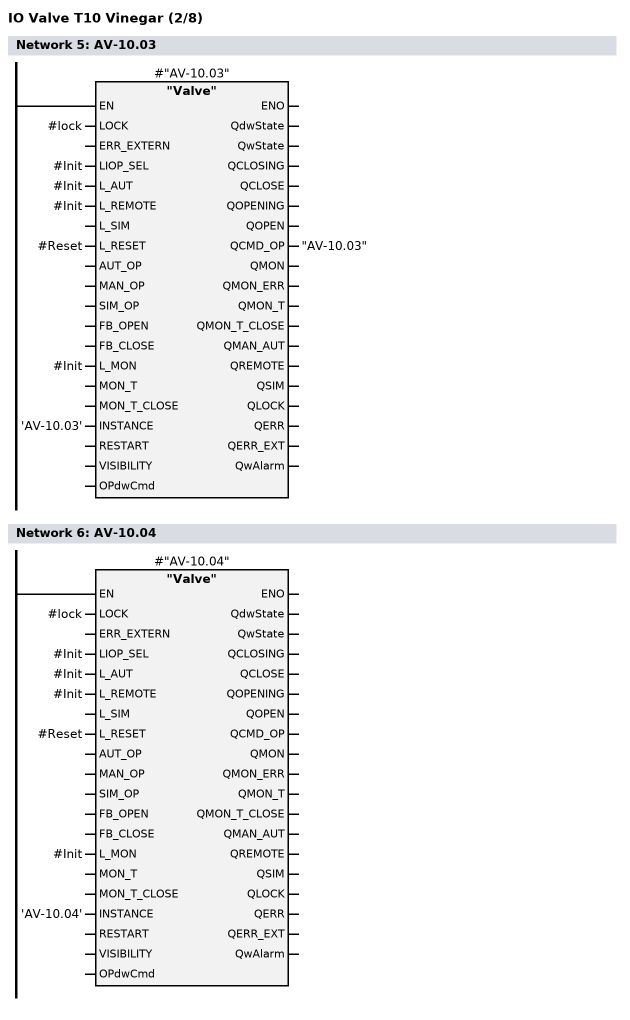
   RUNG wire#powerrail
      #"AV-10.03"(LOCK := #lock, ERR_EXTERN :=, LIOP_SEL := #Init, L_AUT := #Init, L_REMOTE := #Init, L_SIM :=, L_RESET := #Reset, AUT_OP :=, MAN_OP :=, SIM_OP :=, FB_OPEN :=, FB_CLOSE :=, L_MON := #Init, MON_T :=, MON_T_CLOSE :=, INSTANCE := 'AV-10.03', RESTART :=, VISIBILITY :=, OPdwCmd :=, QdwState =>, QwState =>, QCLOSING =>, QCLOSE =>, QOPENING =>, QOPEN =>, QCMD_OP => "AV-10.03", QMON =>, QMON_ERR =>, QMON_T =>, QMON_T_CLOSE =>, QMAN_AUT =>, QREMOTE =>, QSIM =>, QLOCK =>, QERR =>, QERR_EXT =>, QwAlarm =>)
   END_RUNG
   // the same network as SCL:
   #"AV-10.03"(LOCK := #lock,   // "Valve"
               LIOP_SEL := #Init,
               L_AUT := #Init,
               L_REMOTE := #Init,
               L_RESET := #Reset,
               L_MON := #Init,
               INSTANCE := 'AV-10.03',
               QCMD_OP => "AV-10.03");
END_REGION

REGION Network 6: AV-10.04
   RUNG wire#powerrail
      #"AV-10.04"(LOCK := #lock, ERR_EXTERN :=, LIOP_SEL := #Init, L_AUT := #Init, L_REMOTE := #Init, L_SIM :=, L_RESET := #Reset, AUT_OP :=, MAN_OP :=, SIM_OP :=, FB_OPEN :=, FB_CLOSE :=, L_MON := #Init, MON_T :=, MON_T_CLOSE :=, INSTANCE := 'AV-10.04', RESTART :=, VISIBILITY :=, OPdwCmd :=, QdwState =>, QwState =>, QCLOSING =>, QCLOSE =>, QOPENING =>, QOPEN =>, QCMD_OP =>, QMON =>, QMON_ERR =>, QMON_T =>, QMON_T_CLOSE =>, QMAN_AUT =>, QREMOTE =>, QSIM =>, QLOCK =>, QERR =>, QERR_EXT =>, QwAlarm =>)
   END_RUNG
   // the same network as SCL:
   #"AV-10.04"(LOCK := #lock,   // "Valve"
               LIOP_SEL := #Init,
               L_AUT := #Init,
               L_REMOTE := #Init,
               L_RESET := #Reset,
               L_MON := #Init,
               INSTANCE := 'AV-10.04');
END_REGION

REGION Network 7: AV-10.05
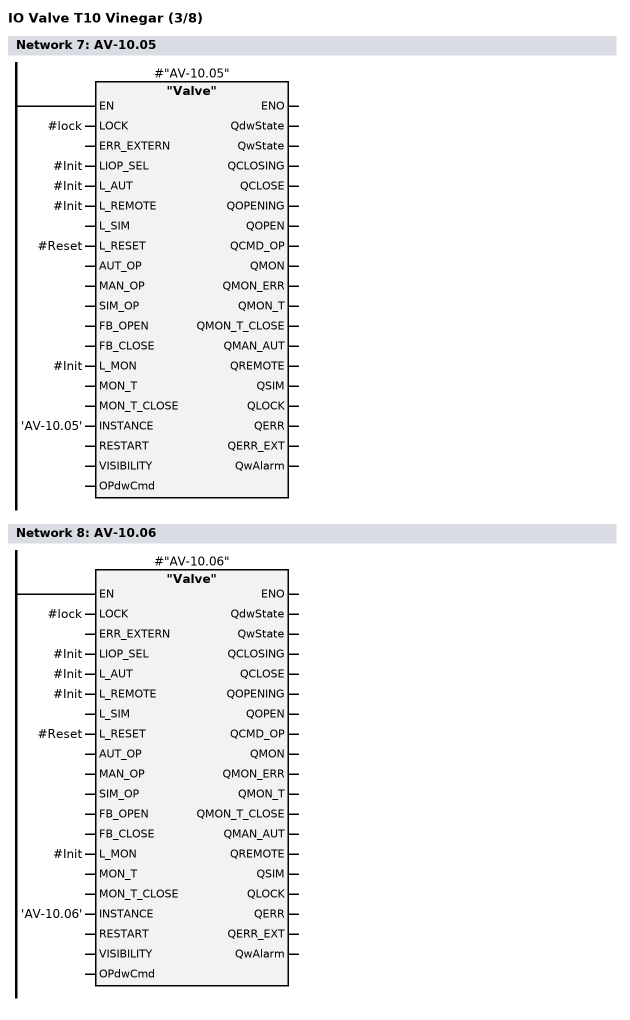
   RUNG wire#powerrail
      #"AV-10.05"(LOCK := #lock, ERR_EXTERN :=, LIOP_SEL := #Init, L_AUT := #Init, L_REMOTE := #Init, L_SIM :=, L_RESET := #Reset, AUT_OP :=, MAN_OP :=, SIM_OP :=, FB_OPEN :=, FB_CLOSE :=, L_MON := #Init, MON_T :=, MON_T_CLOSE :=, INSTANCE := 'AV-10.05', RESTART :=, VISIBILITY :=, OPdwCmd :=, QdwState =>, QwState =>, QCLOSING =>, QCLOSE =>, QOPENING =>, QOPEN =>, QCMD_OP =>, QMON =>, QMON_ERR =>, QMON_T =>, QMON_T_CLOSE =>, QMAN_AUT =>, QREMOTE =>, QSIM =>, QLOCK =>, QERR =>, QERR_EXT =>, QwAlarm =>)
   END_RUNG
   // the same network as SCL:
   #"AV-10.05"(LOCK := #lock,   // "Valve"
               LIOP_SEL := #Init,
               L_AUT := #Init,
               L_REMOTE := #Init,
               L_RESET := #Reset,
               L_MON := #Init,
               INSTANCE := 'AV-10.05');
END_REGION

REGION Network 8: AV-10.06
   RUNG wire#powerrail
      #"AV-10.06"(LOCK := #lock, ERR_EXTERN :=, LIOP_SEL := #Init, L_AUT := #Init, L_REMOTE := #Init, L_SIM :=, L_RESET := #Reset, AUT_OP :=, MAN_OP :=, SIM_OP :=, FB_OPEN :=, FB_CLOSE :=, L_MON := #Init, MON_T :=, MON_T_CLOSE :=, INSTANCE := 'AV-10.06', RESTART :=, VISIBILITY :=, OPdwCmd :=, QdwState =>, QwState =>, QCLOSING =>, QCLOSE =>, QOPENING =>, QOPEN =>, QCMD_OP =>, QMON =>, QMON_ERR =>, QMON_T =>, QMON_T_CLOSE =>, QMAN_AUT =>, QREMOTE =>, QSIM =>, QLOCK =>, QERR =>, QERR_EXT =>, QwAlarm =>)
   END_RUNG
   // the same network as SCL:
   #"AV-10.06"(LOCK := #lock,   // "Valve"
               LIOP_SEL := #Init,
               L_AUT := #Init,
               L_REMOTE := #Init,
               L_RESET := #Reset,
               L_MON := #Init,
               INSTANCE := 'AV-10.06');
END_REGION

REGION Network 9: AV-10.07
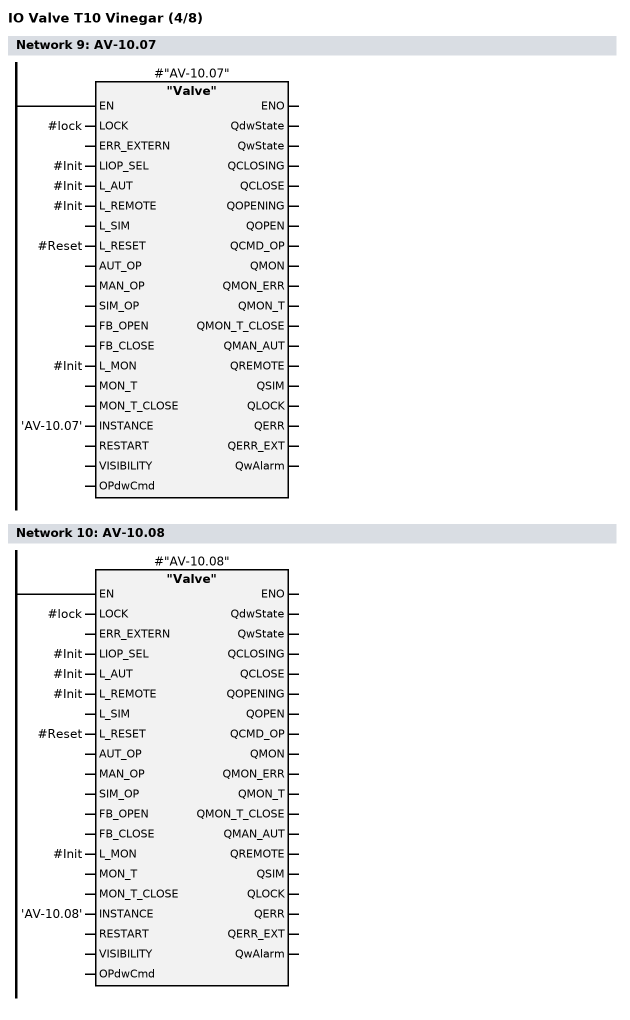
   RUNG wire#powerrail
      #"AV-10.07"(LOCK := #lock, ERR_EXTERN :=, LIOP_SEL := #Init, L_AUT := #Init, L_REMOTE := #Init, L_SIM :=, L_RESET := #Reset, AUT_OP :=, MAN_OP :=, SIM_OP :=, FB_OPEN :=, FB_CLOSE :=, L_MON := #Init, MON_T :=, MON_T_CLOSE :=, INSTANCE := 'AV-10.07', RESTART :=, VISIBILITY :=, OPdwCmd :=, QdwState =>, QwState =>, QCLOSING =>, QCLOSE =>, QOPENING =>, QOPEN =>, QCMD_OP =>, QMON =>, QMON_ERR =>, QMON_T =>, QMON_T_CLOSE =>, QMAN_AUT =>, QREMOTE =>, QSIM =>, QLOCK =>, QERR =>, QERR_EXT =>, QwAlarm =>)
   END_RUNG
   // the same network as SCL:
   #"AV-10.07"(LOCK := #lock,   // "Valve"
               LIOP_SEL := #Init,
               L_AUT := #Init,
               L_REMOTE := #Init,
               L_RESET := #Reset,
               L_MON := #Init,
               INSTANCE := 'AV-10.07');
END_REGION

REGION Network 10: AV-10.08
   RUNG wire#powerrail
      #"AV-10.08"(LOCK := #lock, ERR_EXTERN :=, LIOP_SEL := #Init, L_AUT := #Init, L_REMOTE := #Init, L_SIM :=, L_RESET := #Reset, AUT_OP :=, MAN_OP :=, SIM_OP :=, FB_OPEN :=, FB_CLOSE :=, L_MON := #Init, MON_T :=, MON_T_CLOSE :=, INSTANCE := 'AV-10.08', RESTART :=, VISIBILITY :=, OPdwCmd :=, QdwState =>, QwState =>, QCLOSING =>, QCLOSE =>, QOPENING =>, QOPEN =>, QCMD_OP =>, QMON =>, QMON_ERR =>, QMON_T =>, QMON_T_CLOSE =>, QMAN_AUT =>, QREMOTE =>, QSIM =>, QLOCK =>, QERR =>, QERR_EXT =>, QwAlarm =>)
   END_RUNG
   // the same network as SCL:
   #"AV-10.08"(LOCK := #lock,   // "Valve"
               LIOP_SEL := #Init,
               L_AUT := #Init,
               L_REMOTE := #Init,
               L_RESET := #Reset,
               L_MON := #Init,
               INSTANCE := 'AV-10.08');
END_REGION

REGION Network 11: AV-10.09
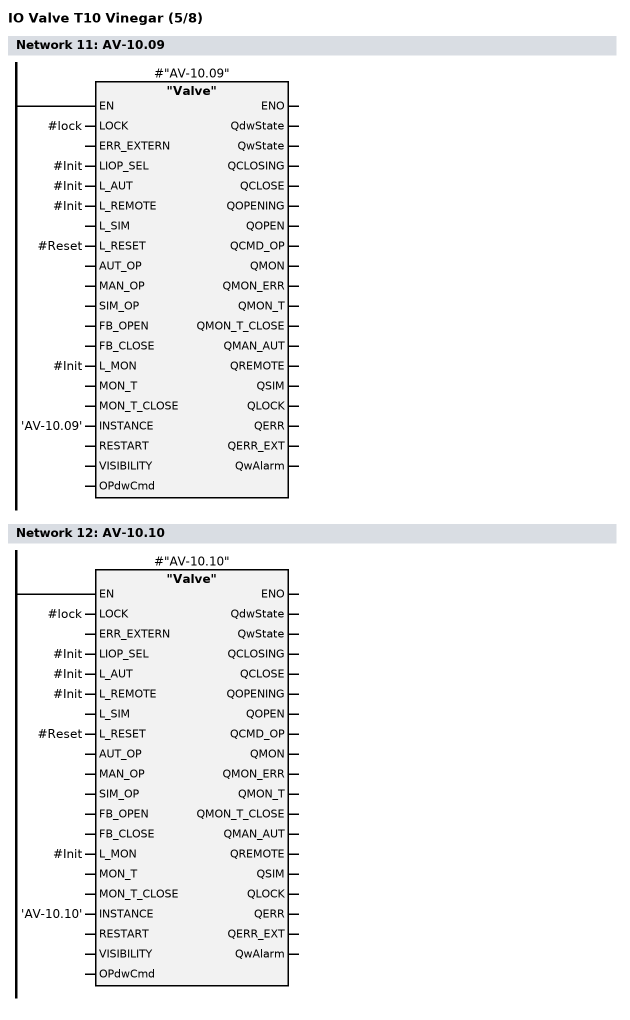
   RUNG wire#powerrail
      #"AV-10.09"(LOCK := #lock, ERR_EXTERN :=, LIOP_SEL := #Init, L_AUT := #Init, L_REMOTE := #Init, L_SIM :=, L_RESET := #Reset, AUT_OP :=, MAN_OP :=, SIM_OP :=, FB_OPEN :=, FB_CLOSE :=, L_MON := #Init, MON_T :=, MON_T_CLOSE :=, INSTANCE := 'AV-10.09', RESTART :=, VISIBILITY :=, OPdwCmd :=, QdwState =>, QwState =>, QCLOSING =>, QCLOSE =>, QOPENING =>, QOPEN =>, QCMD_OP =>, QMON =>, QMON_ERR =>, QMON_T =>, QMON_T_CLOSE =>, QMAN_AUT =>, QREMOTE =>, QSIM =>, QLOCK =>, QERR =>, QERR_EXT =>, QwAlarm =>)
   END_RUNG
   // the same network as SCL:
   #"AV-10.09"(LOCK := #lock,   // "Valve"
               LIOP_SEL := #Init,
               L_AUT := #Init,
               L_REMOTE := #Init,
               L_RESET := #Reset,
               L_MON := #Init,
               INSTANCE := 'AV-10.09');
END_REGION

REGION Network 12: AV-10.10
   RUNG wire#powerrail
      #"AV-10.10"(LOCK := #lock, ERR_EXTERN :=, LIOP_SEL := #Init, L_AUT := #Init, L_REMOTE := #Init, L_SIM :=, L_RESET := #Reset, AUT_OP :=, MAN_OP :=, SIM_OP :=, FB_OPEN :=, FB_CLOSE :=, L_MON := #Init, MON_T :=, MON_T_CLOSE :=, INSTANCE := 'AV-10.10', RESTART :=, VISIBILITY :=, OPdwCmd :=, QdwState =>, QwState =>, QCLOSING =>, QCLOSE =>, QOPENING =>, QOPEN =>, QCMD_OP =>, QMON =>, QMON_ERR =>, QMON_T =>, QMON_T_CLOSE =>, QMAN_AUT =>, QREMOTE =>, QSIM =>, QLOCK =>, QERR =>, QERR_EXT =>, QwAlarm =>)
   END_RUNG
   // the same network as SCL:
   #"AV-10.10"(LOCK := #lock,   // "Valve"
               LIOP_SEL := #Init,
               L_AUT := #Init,
               L_REMOTE := #Init,
               L_RESET := #Reset,
               L_MON := #Init,
               INSTANCE := 'AV-10.10');
END_REGION

REGION Network 13: AV-10.11
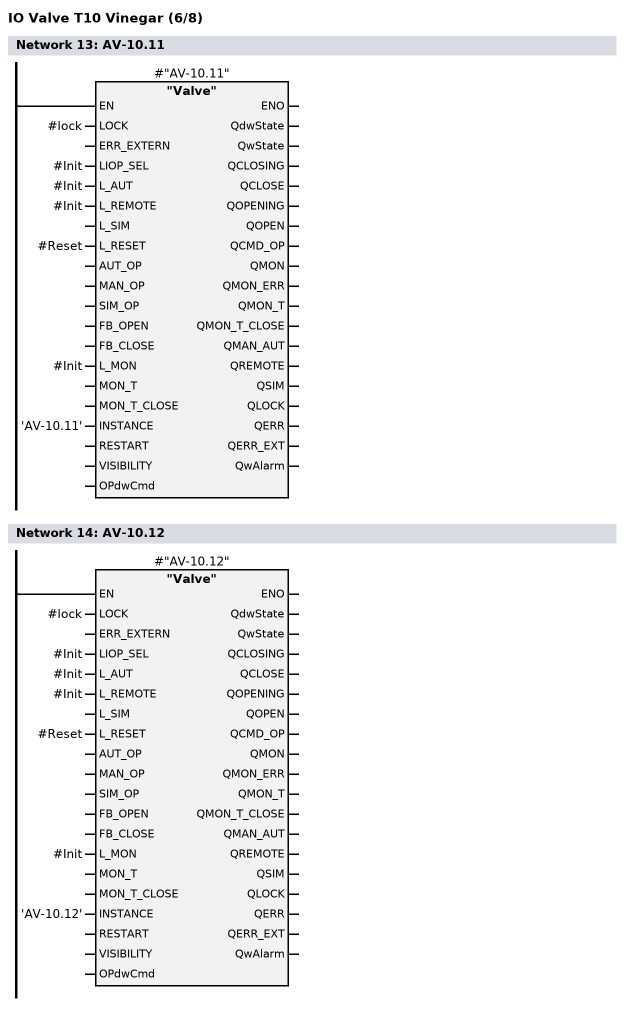
   RUNG wire#powerrail
      #"AV-10.11"(LOCK := #lock, ERR_EXTERN :=, LIOP_SEL := #Init, L_AUT := #Init, L_REMOTE := #Init, L_SIM :=, L_RESET := #Reset, AUT_OP :=, MAN_OP :=, SIM_OP :=, FB_OPEN :=, FB_CLOSE :=, L_MON := #Init, MON_T :=, MON_T_CLOSE :=, INSTANCE := 'AV-10.11', RESTART :=, VISIBILITY :=, OPdwCmd :=, QdwState =>, QwState =>, QCLOSING =>, QCLOSE =>, QOPENING =>, QOPEN =>, QCMD_OP =>, QMON =>, QMON_ERR =>, QMON_T =>, QMON_T_CLOSE =>, QMAN_AUT =>, QREMOTE =>, QSIM =>, QLOCK =>, QERR =>, QERR_EXT =>, QwAlarm =>)
   END_RUNG
   // the same network as SCL:
   #"AV-10.11"(LOCK := #lock,   // "Valve"
               LIOP_SEL := #Init,
               L_AUT := #Init,
               L_REMOTE := #Init,
               L_RESET := #Reset,
               L_MON := #Init,
               INSTANCE := 'AV-10.11');
END_REGION

REGION Network 14: AV-10.12
   RUNG wire#powerrail
      #"AV-10.12"(LOCK := #lock, ERR_EXTERN :=, LIOP_SEL := #Init, L_AUT := #Init, L_REMOTE := #Init, L_SIM :=, L_RESET := #Reset, AUT_OP :=, MAN_OP :=, SIM_OP :=, FB_OPEN :=, FB_CLOSE :=, L_MON := #Init, MON_T :=, MON_T_CLOSE :=, INSTANCE := 'AV-10.12', RESTART :=, VISIBILITY :=, OPdwCmd :=, QdwState =>, QwState =>, QCLOSING =>, QCLOSE =>, QOPENING =>, QOPEN =>, QCMD_OP =>, QMON =>, QMON_ERR =>, QMON_T =>, QMON_T_CLOSE =>, QMAN_AUT =>, QREMOTE =>, QSIM =>, QLOCK =>, QERR =>, QERR_EXT =>, QwAlarm =>)
   END_RUNG
   // the same network as SCL:
   #"AV-10.12"(LOCK := #lock,   // "Valve"
               LIOP_SEL := #Init,
               L_AUT := #Init,
               L_REMOTE := #Init,
               L_RESET := #Reset,
               L_MON := #Init,
               INSTANCE := 'AV-10.12');
END_REGION

REGION Network 15: AV-10.13
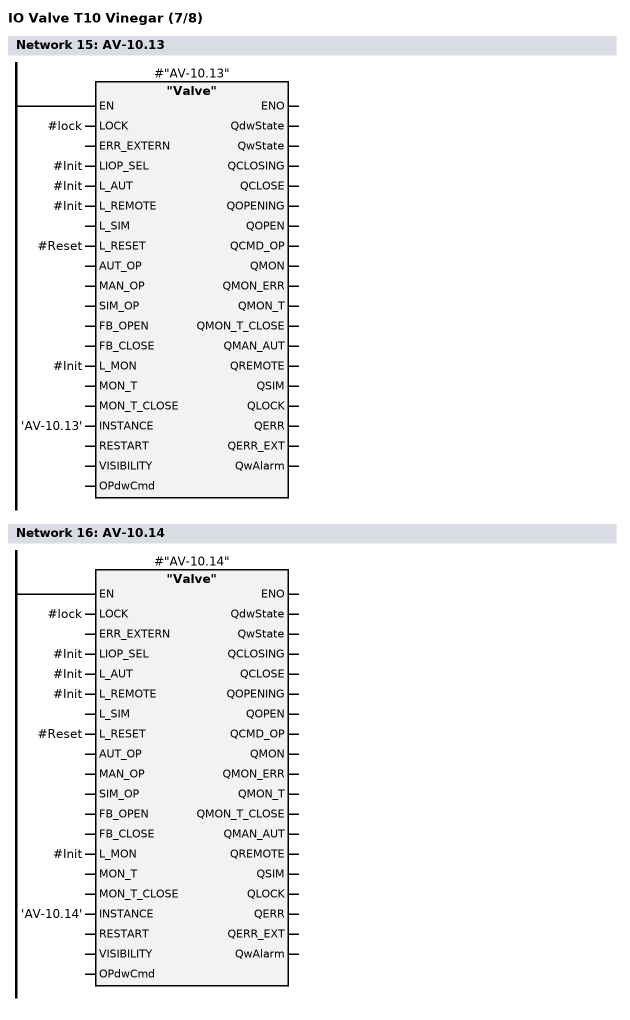
   RUNG wire#powerrail
      #"AV-10.13"(LOCK := #lock, ERR_EXTERN :=, LIOP_SEL := #Init, L_AUT := #Init, L_REMOTE := #Init, L_SIM :=, L_RESET := #Reset, AUT_OP :=, MAN_OP :=, SIM_OP :=, FB_OPEN :=, FB_CLOSE :=, L_MON := #Init, MON_T :=, MON_T_CLOSE :=, INSTANCE := 'AV-10.13', RESTART :=, VISIBILITY :=, OPdwCmd :=, QdwState =>, QwState =>, QCLOSING =>, QCLOSE =>, QOPENING =>, QOPEN =>, QCMD_OP =>, QMON =>, QMON_ERR =>, QMON_T =>, QMON_T_CLOSE =>, QMAN_AUT =>, QREMOTE =>, QSIM =>, QLOCK =>, QERR =>, QERR_EXT =>, QwAlarm =>)
   END_RUNG
   // the same network as SCL:
   #"AV-10.13"(LOCK := #lock,   // "Valve"
               LIOP_SEL := #Init,
               L_AUT := #Init,
               L_REMOTE := #Init,
               L_RESET := #Reset,
               L_MON := #Init,
               INSTANCE := 'AV-10.13');
END_REGION

REGION Network 16: AV-10.14
   RUNG wire#powerrail
      #"AV-10.14"(LOCK := #lock, ERR_EXTERN :=, LIOP_SEL := #Init, L_AUT := #Init, L_REMOTE := #Init, L_SIM :=, L_RESET := #Reset, AUT_OP :=, MAN_OP :=, SIM_OP :=, FB_OPEN :=, FB_CLOSE :=, L_MON := #Init, MON_T :=, MON_T_CLOSE :=, INSTANCE := 'AV-10.14', RESTART :=, VISIBILITY :=, OPdwCmd :=, QdwState =>, QwState =>, QCLOSING =>, QCLOSE =>, QOPENING =>, QOPEN =>, QCMD_OP =>, QMON =>, QMON_ERR =>, QMON_T =>, QMON_T_CLOSE =>, QMAN_AUT =>, QREMOTE =>, QSIM =>, QLOCK =>, QERR =>, QERR_EXT =>, QwAlarm =>)
   END_RUNG
   // the same network as SCL:
   #"AV-10.14"(LOCK := #lock,   // "Valve"
               LIOP_SEL := #Init,
               L_AUT := #Init,
               L_REMOTE := #Init,
               L_RESET := #Reset,
               L_MON := #Init,
               INSTANCE := 'AV-10.14');
END_REGION

REGION Network 17: P-10.02
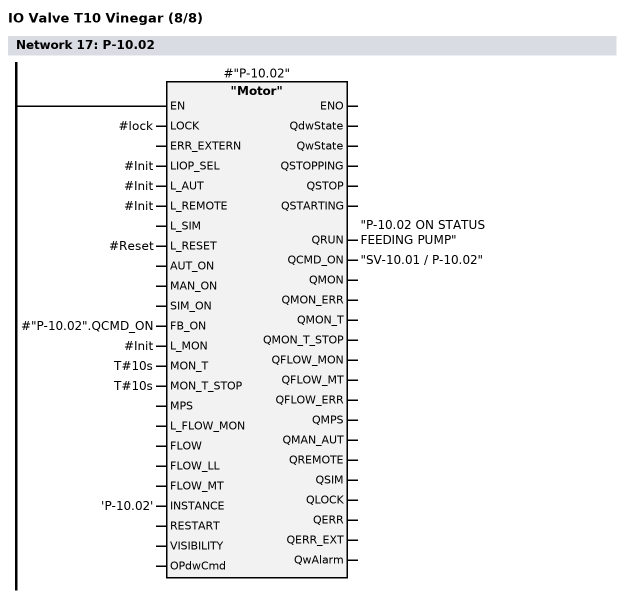
   RUNG wire#powerrail
      #"P-10.02"(LOCK := #lock, ERR_EXTERN :=, LIOP_SEL := #Init, L_AUT := #Init, L_REMOTE := #Init, L_SIM :=, L_RESET := #Reset, AUT_ON :=, MAN_ON :=, SIM_ON :=, FB_ON := #"P-10.02".QCMD_ON, L_MON := #Init, MON_T := T#10s, MON_T_STOP := T#10s, MPS :=, L_FLOW_MON :=, FLOW :=, FLOW_LL :=, FLOW_MT :=, INSTANCE := 'P-10.02', RESTART :=, VISIBILITY :=, OPdwCmd :=, QdwState =>, QwState =>, QSTOPPING =>, QSTOP =>, QSTARTING =>, QRUN => "P-10.02 ON STATUS FEEDING PUMP", QCMD_ON => "SV-10.01 / P-10.02", QMON =>, QMON_ERR =>, QMON_T =>, QMON_T_STOP =>, QFLOW_MON =>, QFLOW_MT =>, QFLOW_ERR =>, QMPS =>, QMAN_AUT =>, QREMOTE =>, QSIM =>, QLOCK =>, QERR =>, QERR_EXT =>, QwAlarm =>)
   END_RUNG
   // the same network as SCL:
   #"P-10.02"(LOCK := #lock,   // "Motor"
              LIOP_SEL := #Init,
              L_AUT := #Init,
              L_REMOTE := #Init,
              L_RESET := #Reset,
              FB_ON := #"P-10.02".QCMD_ON,
              L_MON := #Init,
              MON_T := T#10s,
              MON_T_STOP := T#10s,
              INSTANCE := 'P-10.02',
              QRUN => "P-10.02 ON STATUS FEEDING PUMP",
              QCMD_ON => "SV-10.01 / P-10.02");
END_REGION
END_FUNCTION_BLOCK

FUNCTION_BLOCK "IO Valve T51 HotWaterLine"   // FB311, LAD
{ S7_Optimized_Access := 'FALSE' }
VERSION : 0.1
// stored: AutoNumber false, IsIECCheckEnabled false, SetENOAutomatically false, UDAEnableTagReadback false
   VAR_INPUT
      lock : Bool;
      Init : Bool;
      testing : Bool;
      Reset : Bool;
   END_VAR
   VAR
      "AV-51.01" { S7_SetPoint := 'True'} : "Valve";
      "AV-51.02" { S7_SetPoint := 'True'} : "Valve";
      "AV-51.03" { S7_SetPoint := 'True'} : "Valve";
      "AV-51.04" { S7_SetPoint := 'True'} : "Valve";
      "AV-51.05" { S7_SetPoint := 'True'} : "Valve";
      "AV-51.06" { S7_SetPoint := 'True'} : "Valve";
      "AV-51.07" { S7_SetPoint := 'True'} : "Valve";
      "AV-51.08" { S7_SetPoint := 'True'} : "Valve";
      "AV-51.09" { S7_SetPoint := 'True'} : "Valve";
      "AV-51.10" { S7_SetPoint := 'True'} : "Valve";
      "AV-51.11" { S7_SetPoint := 'True'} : "Valve";
      "AV-51.12" { S7_SetPoint := 'True'} : "Valve";
      "AV-51.13" { S7_SetPoint := 'True'} : "Valve";
      "AV-51.14" { S7_SetPoint := 'True'} : "Valve";
      "AV-51.15" { S7_SetPoint := 'True'} : "Valve";
      "CV-51.11" { S7_SetPoint := 'True'} : "Valve";
   END_VAR
BEGIN

REGION Network 1 (SCL): FB OPEN and CLOSE
   IF #testing THEN
       // Statement section IF
       #"AV-51.01".FB_OPEN := #"AV-51.01".QCMD_OP;
       #"AV-51.01".FB_CLOSE := NOT #"AV-51.01".QCMD_OP;
       #"AV-51.02".FB_OPEN := #"AV-51.02".QCMD_OP;
       #"AV-51.02".FB_CLOSE := NOT #"AV-51.02".QCMD_OP;
       #"AV-51.03".FB_OPEN := #"AV-51.03".QCMD_OP;
       #"AV-51.03".FB_CLOSE := NOT #"AV-51.03".QCMD_OP;
       #"AV-51.04".FB_OPEN := #"AV-51.04".QCMD_OP;
       #"AV-51.04".FB_CLOSE := NOT #"AV-51.04".QCMD_OP;
       #"AV-51.05".FB_OPEN := #"AV-51.05".QCMD_OP;
       #"AV-51.05".FB_CLOSE := NOT #"AV-51.05".QCMD_OP;
       #"AV-51.06".FB_OPEN := #"AV-51.06".QCMD_OP;
       #"AV-51.06".FB_CLOSE := NOT #"AV-51.06".QCMD_OP;
       #"AV-51.07".FB_OPEN := #"AV-51.07".QCMD_OP;
       #"AV-51.07".FB_CLOSE := NOT #"AV-51.07".QCMD_OP;
       #"AV-51.08".FB_OPEN := #"AV-51.08".QCMD_OP;
       #"AV-51.08".FB_CLOSE := NOT #"AV-51.08".QCMD_OP;
       #"AV-51.09".FB_OPEN := #"AV-51.09".QCMD_OP;
       #"AV-51.09".FB_CLOSE := NOT #"AV-51.09".QCMD_OP;
       #"AV-51.10".FB_OPEN := #"AV-51.10".QCMD_OP;
       #"AV-51.10".FB_CLOSE := NOT #"AV-51.10".QCMD_OP;
       #"AV-51.11".FB_OPEN := #"AV-51.11".QCMD_OP;
       #"AV-51.11".FB_CLOSE := NOT #"AV-51.11".QCMD_OP;
       #"AV-51.12".FB_OPEN := #"AV-51.12".QCMD_OP;
       #"AV-51.12".FB_CLOSE := NOT #"AV-51.12".QCMD_OP;
       #"AV-51.13".FB_OPEN := #"AV-51.13".QCMD_OP;
       #"AV-51.13".FB_CLOSE := NOT #"AV-51.13".QCMD_OP;
       #"AV-51.14".FB_OPEN := #"AV-51.14".QCMD_OP;
       #"AV-51.14".FB_CLOSE := NOT #"AV-51.14".QCMD_OP;
       #"AV-51.15".FB_OPEN := #"AV-51.15".QCMD_OP;
       #"AV-51.15".FB_CLOSE := NOT #"AV-51.15".QCMD_OP;
   ELSE
       // Statement section ELSE
       #"AV-51.01".FB_OPEN := #"AV-51.01".QCMD_OP;
       #"AV-51.01".FB_CLOSE := NOT #"AV-51.01".QCMD_OP;
       #"AV-51.02".FB_OPEN := #"AV-51.02".QCMD_OP;
       #"AV-51.02".FB_CLOSE := NOT #"AV-51.02".QCMD_OP;
       #"AV-51.03".FB_OPEN := #"AV-51.03".QCMD_OP;
       #"AV-51.03".FB_CLOSE := NOT #"AV-51.03".QCMD_OP;
       #"AV-51.04".FB_OPEN := NOT "ZSC-51.04";
       #"AV-51.04".FB_CLOSE := "ZSC-51.04";
       #"AV-51.05".FB_OPEN := NOT "ZSC-51.05";
       #"AV-51.05".FB_CLOSE := "ZSC-51.05";
       #"AV-51.06".FB_OPEN := #"AV-51.06".QCMD_OP;
       #"AV-51.06".FB_CLOSE := NOT #"AV-51.06".QCMD_OP;
       #"AV-51.07".FB_OPEN := #"AV-51.07".QCMD_OP;
       #"AV-51.07".FB_CLOSE := NOT #"AV-51.07".QCMD_OP;
       #"AV-51.08".FB_OPEN := #"AV-51.08".QCMD_OP;
       #"AV-51.08".FB_CLOSE := NOT #"AV-51.08".QCMD_OP;
       #"AV-51.09".FB_OPEN := #"AV-51.09".QCMD_OP;
       #"AV-51.09".FB_CLOSE := NOT #"AV-51.09".QCMD_OP;
       #"AV-51.10".FB_OPEN := #"AV-51.10".QCMD_OP;
       #"AV-51.10".FB_CLOSE := NOT #"AV-51.10".QCMD_OP;
       #"AV-51.11".FB_OPEN := #"AV-51.11".QCMD_OP;
       #"AV-51.11".FB_CLOSE := NOT #"AV-51.11".QCMD_OP;
       #"AV-51.12".FB_OPEN := #"AV-51.12".QCMD_OP;
       #"AV-51.12".FB_CLOSE := NOT #"AV-51.12".QCMD_OP;
       #"AV-51.13".FB_OPEN := #"AV-51.13".QCMD_OP;
       #"AV-51.13".FB_CLOSE := NOT #"AV-51.13".QCMD_OP;
       #"AV-51.14".FB_OPEN := #"AV-51.14".QCMD_OP;
       #"AV-51.14".FB_CLOSE := NOT #"AV-51.14".QCMD_OP;
       #"AV-51.15".FB_OPEN := #"AV-51.15".QCMD_OP;
       #"AV-51.15".FB_CLOSE := NOT #"AV-51.15".QCMD_OP;
   END_IF;
END_REGION

NETWORK
TITLE = FB Monitoring Time
// FB OPEN Time
      L     t#20s;
      T     #"AV-51.01".MON_T;
      T     #"AV-51.02".MON_T;
      T     #"AV-51.03".MON_T;
      T     #"AV-51.04".MON_T;
      T     #"AV-51.05".MON_T;
      T     #"AV-51.06".MON_T;
      T     #"AV-51.07".MON_T;
      T     #"AV-51.08".MON_T;
      T     #"AV-51.09".MON_T;
      T     #"AV-51.10".MON_T;
      T     #"AV-51.11".MON_T;
      T     #"AV-51.12".MON_T;
      T     #"AV-51.13".MON_T;
      T     #"AV-51.14".MON_T;
      T     #"AV-51.15".MON_T;
// FB CLOSE Time
      L     t#20s;
      T     #"AV-51.01".MON_T_CLOSE;
      T     #"AV-51.02".MON_T_CLOSE;
      T     #"AV-51.03".MON_T_CLOSE;
      T     #"AV-51.04".MON_T_CLOSE;
      T     #"AV-51.05".MON_T_CLOSE;
      T     #"AV-51.06".MON_T_CLOSE;
      T     #"AV-51.07".MON_T_CLOSE;
      T     #"AV-51.08".MON_T_CLOSE;
      T     #"AV-51.09".MON_T_CLOSE;
      T     #"AV-51.10".MON_T_CLOSE;
      T     #"AV-51.11".MON_T_CLOSE;
      T     #"AV-51.12".MON_T_CLOSE;
      T     #"AV-51.13".MON_T_CLOSE;
      T     #"AV-51.14".MON_T_CLOSE;
      T     #"AV-51.15".MON_T_CLOSE;

REGION Network 3: AV-51.01
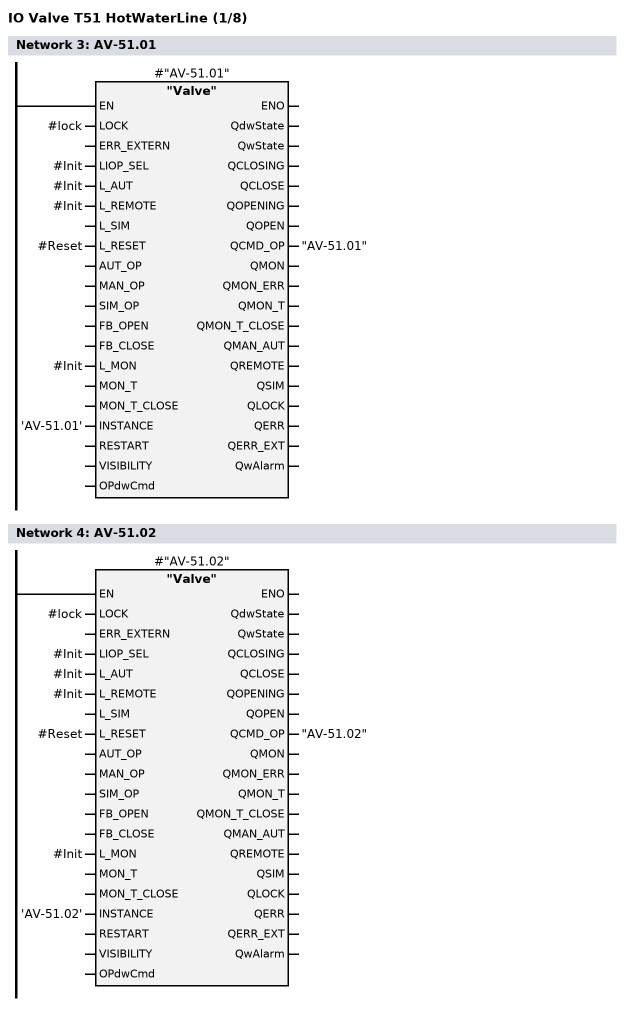
   RUNG wire#powerrail
      #"AV-51.01"(LOCK := #lock, ERR_EXTERN :=, LIOP_SEL := #Init, L_AUT := #Init, L_REMOTE := #Init, L_SIM :=, L_RESET := #Reset, AUT_OP :=, MAN_OP :=, SIM_OP :=, FB_OPEN :=, FB_CLOSE :=, L_MON := #Init, MON_T :=, MON_T_CLOSE :=, INSTANCE := 'AV-51.01', RESTART :=, VISIBILITY :=, OPdwCmd :=, QdwState =>, QwState =>, QCLOSING =>, QCLOSE =>, QOPENING =>, QOPEN =>, QCMD_OP => "AV-51.01", QMON =>, QMON_ERR =>, QMON_T =>, QMON_T_CLOSE =>, QMAN_AUT =>, QREMOTE =>, QSIM =>, QLOCK =>, QERR =>, QERR_EXT =>, QwAlarm =>)
   END_RUNG
   // the same network as SCL:
   #"AV-51.01"(LOCK := #lock,   // "Valve"
               LIOP_SEL := #Init,
               L_AUT := #Init,
               L_REMOTE := #Init,
               L_RESET := #Reset,
               L_MON := #Init,
               INSTANCE := 'AV-51.01',
               QCMD_OP => "AV-51.01");
END_REGION

REGION Network 4: AV-51.02
   RUNG wire#powerrail
      #"AV-51.02"(LOCK := #lock, ERR_EXTERN :=, LIOP_SEL := #Init, L_AUT := #Init, L_REMOTE := #Init, L_SIM :=, L_RESET := #Reset, AUT_OP :=, MAN_OP :=, SIM_OP :=, FB_OPEN :=, FB_CLOSE :=, L_MON := #Init, MON_T :=, MON_T_CLOSE :=, INSTANCE := 'AV-51.02', RESTART :=, VISIBILITY :=, OPdwCmd :=, QdwState =>, QwState =>, QCLOSING =>, QCLOSE =>, QOPENING =>, QOPEN =>, QCMD_OP => "AV-51.02", QMON =>, QMON_ERR =>, QMON_T =>, QMON_T_CLOSE =>, QMAN_AUT =>, QREMOTE =>, QSIM =>, QLOCK =>, QERR =>, QERR_EXT =>, QwAlarm =>)
   END_RUNG
   // the same network as SCL:
   #"AV-51.02"(LOCK := #lock,   // "Valve"
               LIOP_SEL := #Init,
               L_AUT := #Init,
               L_REMOTE := #Init,
               L_RESET := #Reset,
               L_MON := #Init,
               INSTANCE := 'AV-51.02',
               QCMD_OP => "AV-51.02");
END_REGION

REGION Network 5: AV-51.03
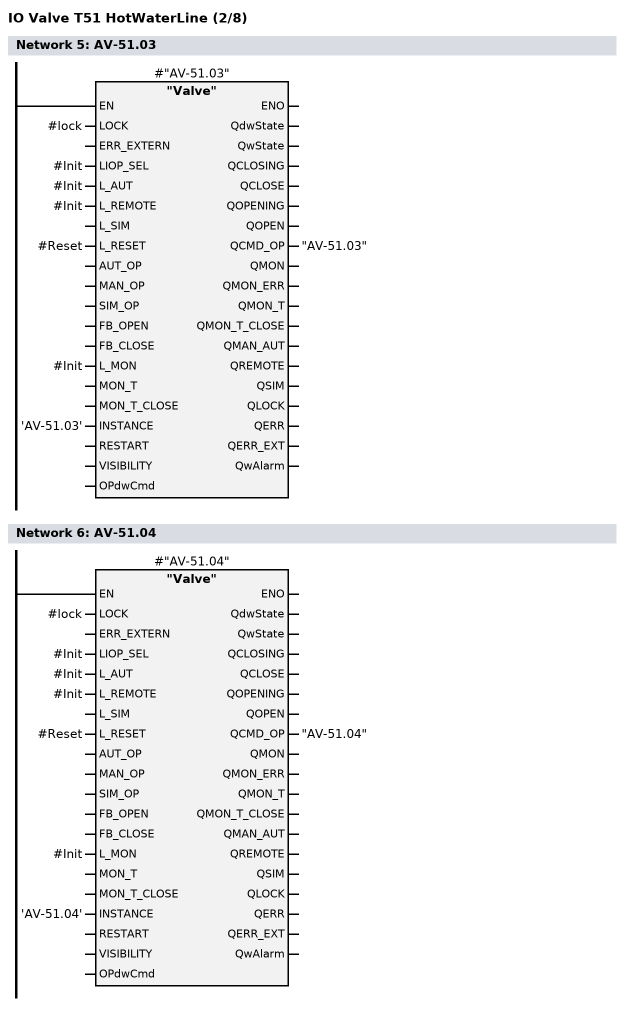
   RUNG wire#powerrail
      #"AV-51.03"(LOCK := #lock, ERR_EXTERN :=, LIOP_SEL := #Init, L_AUT := #Init, L_REMOTE := #Init, L_SIM :=, L_RESET := #Reset, AUT_OP :=, MAN_OP :=, SIM_OP :=, FB_OPEN :=, FB_CLOSE :=, L_MON := #Init, MON_T :=, MON_T_CLOSE :=, INSTANCE := 'AV-51.03', RESTART :=, VISIBILITY :=, OPdwCmd :=, QdwState =>, QwState =>, QCLOSING =>, QCLOSE =>, QOPENING =>, QOPEN =>, QCMD_OP => "AV-51.03", QMON =>, QMON_ERR =>, QMON_T =>, QMON_T_CLOSE =>, QMAN_AUT =>, QREMOTE =>, QSIM =>, QLOCK =>, QERR =>, QERR_EXT =>, QwAlarm =>)
   END_RUNG
   // the same network as SCL:
   #"AV-51.03"(LOCK := #lock,   // "Valve"
               LIOP_SEL := #Init,
               L_AUT := #Init,
               L_REMOTE := #Init,
               L_RESET := #Reset,
               L_MON := #Init,
               INSTANCE := 'AV-51.03',
               QCMD_OP => "AV-51.03");
END_REGION

REGION Network 6: AV-51.04
   RUNG wire#powerrail
      #"AV-51.04"(LOCK := #lock, ERR_EXTERN :=, LIOP_SEL := #Init, L_AUT := #Init, L_REMOTE := #Init, L_SIM :=, L_RESET := #Reset, AUT_OP :=, MAN_OP :=, SIM_OP :=, FB_OPEN :=, FB_CLOSE :=, L_MON := #Init, MON_T :=, MON_T_CLOSE :=, INSTANCE := 'AV-51.04', RESTART :=, VISIBILITY :=, OPdwCmd :=, QdwState =>, QwState =>, QCLOSING =>, QCLOSE =>, QOPENING =>, QOPEN =>, QCMD_OP => "AV-51.04", QMON =>, QMON_ERR =>, QMON_T =>, QMON_T_CLOSE =>, QMAN_AUT =>, QREMOTE =>, QSIM =>, QLOCK =>, QERR =>, QERR_EXT =>, QwAlarm =>)
   END_RUNG
   // the same network as SCL:
   #"AV-51.04"(LOCK := #lock,   // "Valve"
               LIOP_SEL := #Init,
               L_AUT := #Init,
               L_REMOTE := #Init,
               L_RESET := #Reset,
               L_MON := #Init,
               INSTANCE := 'AV-51.04',
               QCMD_OP => "AV-51.04");
END_REGION

REGION Network 7: AV-51.05
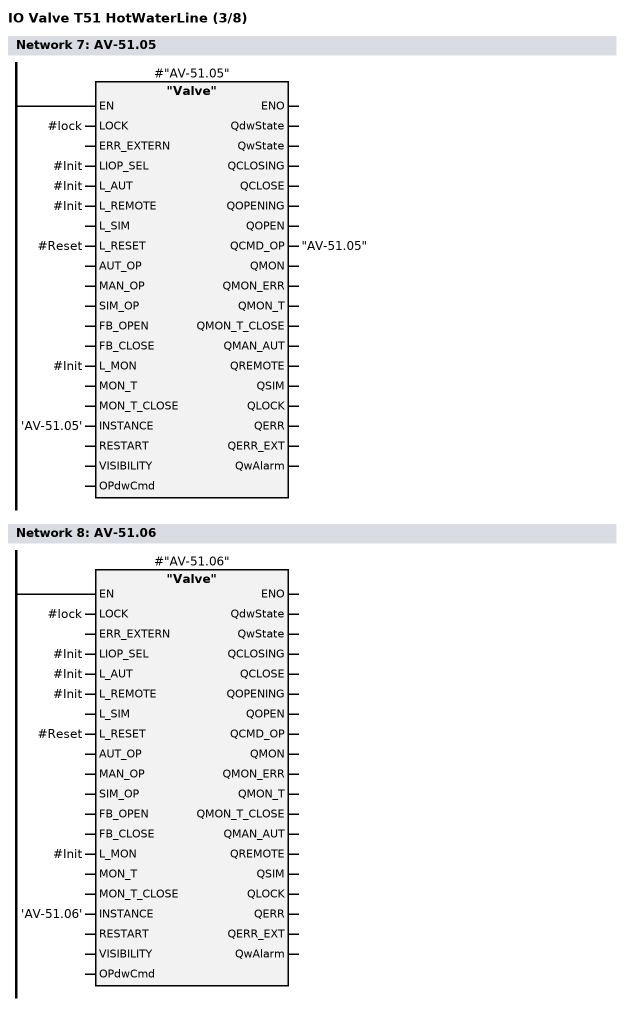
   RUNG wire#powerrail
      #"AV-51.05"(LOCK := #lock, ERR_EXTERN :=, LIOP_SEL := #Init, L_AUT := #Init, L_REMOTE := #Init, L_SIM :=, L_RESET := #Reset, AUT_OP :=, MAN_OP :=, SIM_OP :=, FB_OPEN :=, FB_CLOSE :=, L_MON := #Init, MON_T :=, MON_T_CLOSE :=, INSTANCE := 'AV-51.05', RESTART :=, VISIBILITY :=, OPdwCmd :=, QdwState =>, QwState =>, QCLOSING =>, QCLOSE =>, QOPENING =>, QOPEN =>, QCMD_OP => "AV-51.05", QMON =>, QMON_ERR =>, QMON_T =>, QMON_T_CLOSE =>, QMAN_AUT =>, QREMOTE =>, QSIM =>, QLOCK =>, QERR =>, QERR_EXT =>, QwAlarm =>)
   END_RUNG
   // the same network as SCL:
   #"AV-51.05"(LOCK := #lock,   // "Valve"
               LIOP_SEL := #Init,
               L_AUT := #Init,
               L_REMOTE := #Init,
               L_RESET := #Reset,
               L_MON := #Init,
               INSTANCE := 'AV-51.05',
               QCMD_OP => "AV-51.05");
END_REGION

REGION Network 8: AV-51.06
   RUNG wire#powerrail
      #"AV-51.06"(LOCK := #lock, ERR_EXTERN :=, LIOP_SEL := #Init, L_AUT := #Init, L_REMOTE := #Init, L_SIM :=, L_RESET := #Reset, AUT_OP :=, MAN_OP :=, SIM_OP :=, FB_OPEN :=, FB_CLOSE :=, L_MON := #Init, MON_T :=, MON_T_CLOSE :=, INSTANCE := 'AV-51.06', RESTART :=, VISIBILITY :=, OPdwCmd :=, QdwState =>, QwState =>, QCLOSING =>, QCLOSE =>, QOPENING =>, QOPEN =>, QCMD_OP =>, QMON =>, QMON_ERR =>, QMON_T =>, QMON_T_CLOSE =>, QMAN_AUT =>, QREMOTE =>, QSIM =>, QLOCK =>, QERR =>, QERR_EXT =>, QwAlarm =>)
   END_RUNG
   // the same network as SCL:
   #"AV-51.06"(LOCK := #lock,   // "Valve"
               LIOP_SEL := #Init,
               L_AUT := #Init,
               L_REMOTE := #Init,
               L_RESET := #Reset,
               L_MON := #Init,
               INSTANCE := 'AV-51.06');
END_REGION

REGION Network 9: AV-51.07
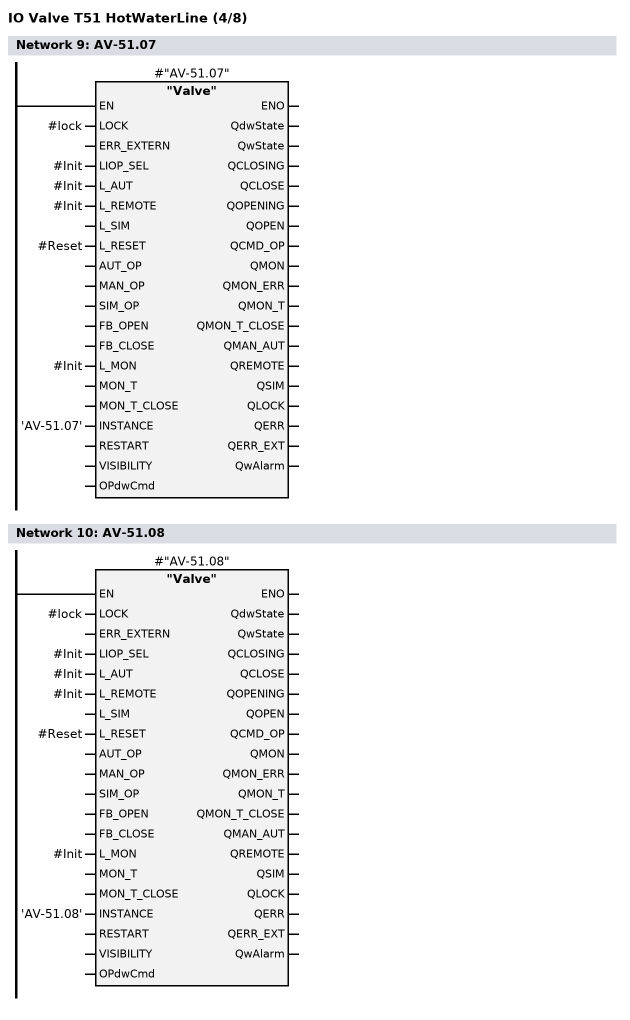
   RUNG wire#powerrail
      #"AV-51.07"(LOCK := #lock, ERR_EXTERN :=, LIOP_SEL := #Init, L_AUT := #Init, L_REMOTE := #Init, L_SIM :=, L_RESET := #Reset, AUT_OP :=, MAN_OP :=, SIM_OP :=, FB_OPEN :=, FB_CLOSE :=, L_MON := #Init, MON_T :=, MON_T_CLOSE :=, INSTANCE := 'AV-51.07', RESTART :=, VISIBILITY :=, OPdwCmd :=, QdwState =>, QwState =>, QCLOSING =>, QCLOSE =>, QOPENING =>, QOPEN =>, QCMD_OP =>, QMON =>, QMON_ERR =>, QMON_T =>, QMON_T_CLOSE =>, QMAN_AUT =>, QREMOTE =>, QSIM =>, QLOCK =>, QERR =>, QERR_EXT =>, QwAlarm =>)
   END_RUNG
   // the same network as SCL:
   #"AV-51.07"(LOCK := #lock,   // "Valve"
               LIOP_SEL := #Init,
               L_AUT := #Init,
               L_REMOTE := #Init,
               L_RESET := #Reset,
               L_MON := #Init,
               INSTANCE := 'AV-51.07');
END_REGION

REGION Network 10: AV-51.08
   RUNG wire#powerrail
      #"AV-51.08"(LOCK := #lock, ERR_EXTERN :=, LIOP_SEL := #Init, L_AUT := #Init, L_REMOTE := #Init, L_SIM :=, L_RESET := #Reset, AUT_OP :=, MAN_OP :=, SIM_OP :=, FB_OPEN :=, FB_CLOSE :=, L_MON := #Init, MON_T :=, MON_T_CLOSE :=, INSTANCE := 'AV-51.08', RESTART :=, VISIBILITY :=, OPdwCmd :=, QdwState =>, QwState =>, QCLOSING =>, QCLOSE =>, QOPENING =>, QOPEN =>, QCMD_OP =>, QMON =>, QMON_ERR =>, QMON_T =>, QMON_T_CLOSE =>, QMAN_AUT =>, QREMOTE =>, QSIM =>, QLOCK =>, QERR =>, QERR_EXT =>, QwAlarm =>)
   END_RUNG
   // the same network as SCL:
   #"AV-51.08"(LOCK := #lock,   // "Valve"
               LIOP_SEL := #Init,
               L_AUT := #Init,
               L_REMOTE := #Init,
               L_RESET := #Reset,
               L_MON := #Init,
               INSTANCE := 'AV-51.08');
END_REGION

REGION Network 11: AV-51.09
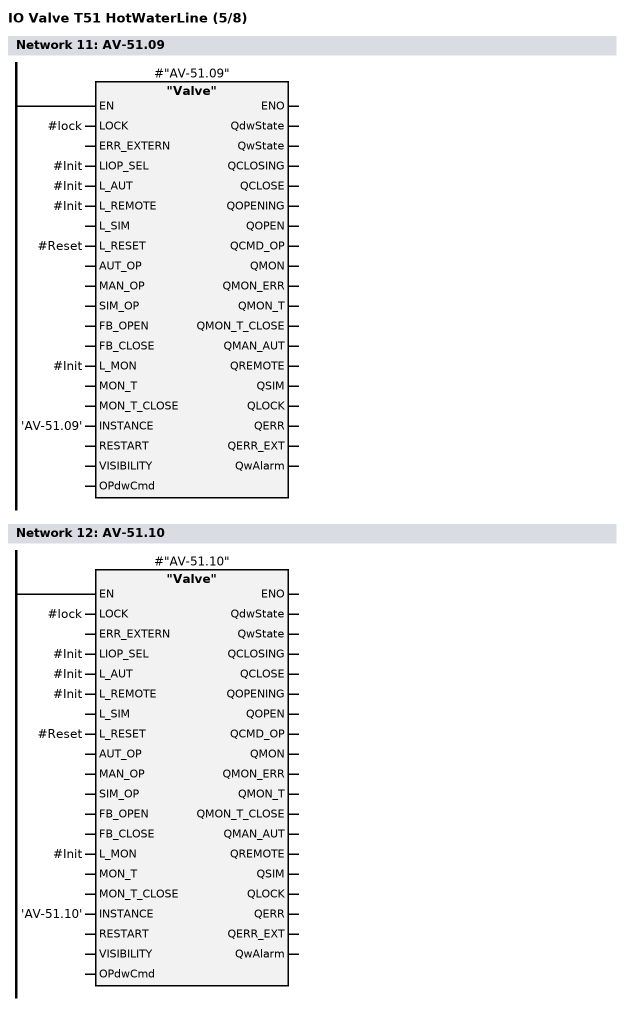
   RUNG wire#powerrail
      #"AV-51.09"(LOCK := #lock, ERR_EXTERN :=, LIOP_SEL := #Init, L_AUT := #Init, L_REMOTE := #Init, L_SIM :=, L_RESET := #Reset, AUT_OP :=, MAN_OP :=, SIM_OP :=, FB_OPEN :=, FB_CLOSE :=, L_MON := #Init, MON_T :=, MON_T_CLOSE :=, INSTANCE := 'AV-51.09', RESTART :=, VISIBILITY :=, OPdwCmd :=, QdwState =>, QwState =>, QCLOSING =>, QCLOSE =>, QOPENING =>, QOPEN =>, QCMD_OP =>, QMON =>, QMON_ERR =>, QMON_T =>, QMON_T_CLOSE =>, QMAN_AUT =>, QREMOTE =>, QSIM =>, QLOCK =>, QERR =>, QERR_EXT =>, QwAlarm =>)
   END_RUNG
   // the same network as SCL:
   #"AV-51.09"(LOCK := #lock,   // "Valve"
               LIOP_SEL := #Init,
               L_AUT := #Init,
               L_REMOTE := #Init,
               L_RESET := #Reset,
               L_MON := #Init,
               INSTANCE := 'AV-51.09');
END_REGION

REGION Network 12: AV-51.10
   RUNG wire#powerrail
      #"AV-51.10"(LOCK := #lock, ERR_EXTERN :=, LIOP_SEL := #Init, L_AUT := #Init, L_REMOTE := #Init, L_SIM :=, L_RESET := #Reset, AUT_OP :=, MAN_OP :=, SIM_OP :=, FB_OPEN :=, FB_CLOSE :=, L_MON := #Init, MON_T :=, MON_T_CLOSE :=, INSTANCE := 'AV-51.10', RESTART :=, VISIBILITY :=, OPdwCmd :=, QdwState =>, QwState =>, QCLOSING =>, QCLOSE =>, QOPENING =>, QOPEN =>, QCMD_OP =>, QMON =>, QMON_ERR =>, QMON_T =>, QMON_T_CLOSE =>, QMAN_AUT =>, QREMOTE =>, QSIM =>, QLOCK =>, QERR =>, QERR_EXT =>, QwAlarm =>)
   END_RUNG
   // the same network as SCL:
   #"AV-51.10"(LOCK := #lock,   // "Valve"
               LIOP_SEL := #Init,
               L_AUT := #Init,
               L_REMOTE := #Init,
               L_RESET := #Reset,
               L_MON := #Init,
               INSTANCE := 'AV-51.10');
END_REGION

REGION Network 13: AV-51.11
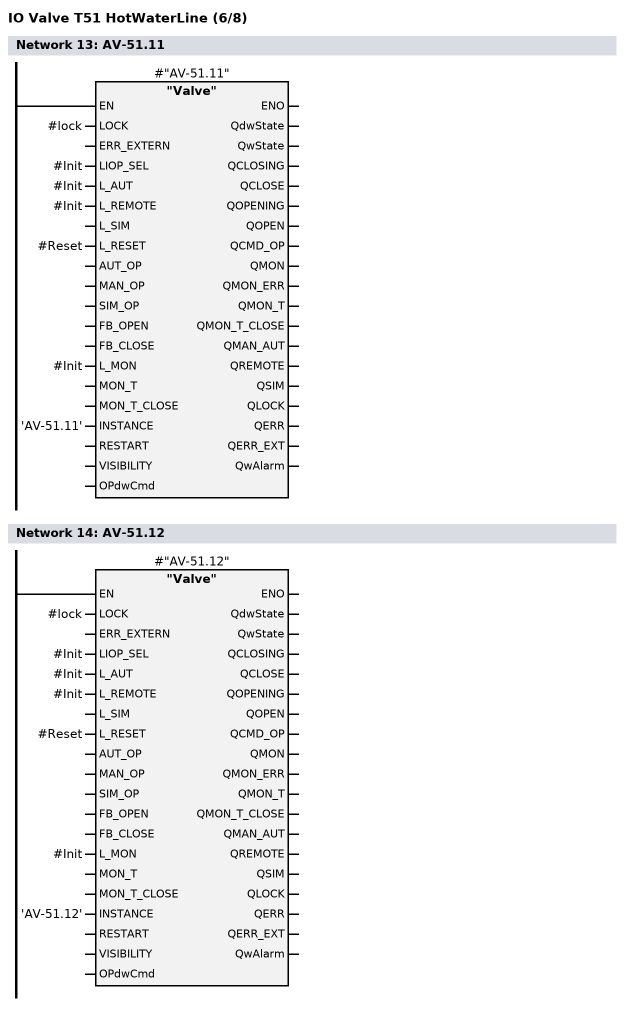
   RUNG wire#powerrail
      #"AV-51.11"(LOCK := #lock, ERR_EXTERN :=, LIOP_SEL := #Init, L_AUT := #Init, L_REMOTE := #Init, L_SIM :=, L_RESET := #Reset, AUT_OP :=, MAN_OP :=, SIM_OP :=, FB_OPEN :=, FB_CLOSE :=, L_MON := #Init, MON_T :=, MON_T_CLOSE :=, INSTANCE := 'AV-51.11', RESTART :=, VISIBILITY :=, OPdwCmd :=, QdwState =>, QwState =>, QCLOSING =>, QCLOSE =>, QOPENING =>, QOPEN =>, QCMD_OP =>, QMON =>, QMON_ERR =>, QMON_T =>, QMON_T_CLOSE =>, QMAN_AUT =>, QREMOTE =>, QSIM =>, QLOCK =>, QERR =>, QERR_EXT =>, QwAlarm =>)
   END_RUNG
   // the same network as SCL:
   #"AV-51.11"(LOCK := #lock,   // "Valve"
               LIOP_SEL := #Init,
               L_AUT := #Init,
               L_REMOTE := #Init,
               L_RESET := #Reset,
               L_MON := #Init,
               INSTANCE := 'AV-51.11');
END_REGION

REGION Network 14: AV-51.12
   RUNG wire#powerrail
      #"AV-51.12"(LOCK := #lock, ERR_EXTERN :=, LIOP_SEL := #Init, L_AUT := #Init, L_REMOTE := #Init, L_SIM :=, L_RESET := #Reset, AUT_OP :=, MAN_OP :=, SIM_OP :=, FB_OPEN :=, FB_CLOSE :=, L_MON := #Init, MON_T :=, MON_T_CLOSE :=, INSTANCE := 'AV-51.12', RESTART :=, VISIBILITY :=, OPdwCmd :=, QdwState =>, QwState =>, QCLOSING =>, QCLOSE =>, QOPENING =>, QOPEN =>, QCMD_OP =>, QMON =>, QMON_ERR =>, QMON_T =>, QMON_T_CLOSE =>, QMAN_AUT =>, QREMOTE =>, QSIM =>, QLOCK =>, QERR =>, QERR_EXT =>, QwAlarm =>)
   END_RUNG
   // the same network as SCL:
   #"AV-51.12"(LOCK := #lock,   // "Valve"
               LIOP_SEL := #Init,
               L_AUT := #Init,
               L_REMOTE := #Init,
               L_RESET := #Reset,
               L_MON := #Init,
               INSTANCE := 'AV-51.12');
END_REGION

REGION Network 15: AV-51.13
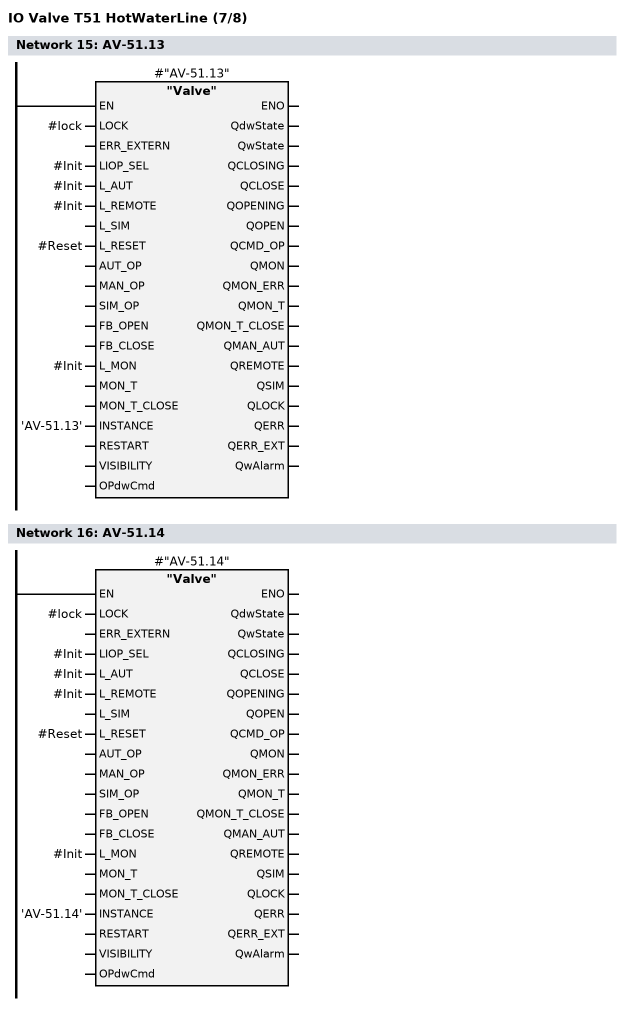
   RUNG wire#powerrail
      #"AV-51.13"(LOCK := #lock, ERR_EXTERN :=, LIOP_SEL := #Init, L_AUT := #Init, L_REMOTE := #Init, L_SIM :=, L_RESET := #Reset, AUT_OP :=, MAN_OP :=, SIM_OP :=, FB_OPEN :=, FB_CLOSE :=, L_MON := #Init, MON_T :=, MON_T_CLOSE :=, INSTANCE := 'AV-51.13', RESTART :=, VISIBILITY :=, OPdwCmd :=, QdwState =>, QwState =>, QCLOSING =>, QCLOSE =>, QOPENING =>, QOPEN =>, QCMD_OP =>, QMON =>, QMON_ERR =>, QMON_T =>, QMON_T_CLOSE =>, QMAN_AUT =>, QREMOTE =>, QSIM =>, QLOCK =>, QERR =>, QERR_EXT =>, QwAlarm =>)
   END_RUNG
   // the same network as SCL:
   #"AV-51.13"(LOCK := #lock,   // "Valve"
               LIOP_SEL := #Init,
               L_AUT := #Init,
               L_REMOTE := #Init,
               L_RESET := #Reset,
               L_MON := #Init,
               INSTANCE := 'AV-51.13');
END_REGION

REGION Network 16: AV-51.14
   RUNG wire#powerrail
      #"AV-51.14"(LOCK := #lock, ERR_EXTERN :=, LIOP_SEL := #Init, L_AUT := #Init, L_REMOTE := #Init, L_SIM :=, L_RESET := #Reset, AUT_OP :=, MAN_OP :=, SIM_OP :=, FB_OPEN :=, FB_CLOSE :=, L_MON := #Init, MON_T :=, MON_T_CLOSE :=, INSTANCE := 'AV-51.14', RESTART :=, VISIBILITY :=, OPdwCmd :=, QdwState =>, QwState =>, QCLOSING =>, QCLOSE =>, QOPENING =>, QOPEN =>, QCMD_OP =>, QMON =>, QMON_ERR =>, QMON_T =>, QMON_T_CLOSE =>, QMAN_AUT =>, QREMOTE =>, QSIM =>, QLOCK =>, QERR =>, QERR_EXT =>, QwAlarm =>)
   END_RUNG
   // the same network as SCL:
   #"AV-51.14"(LOCK := #lock,   // "Valve"
               LIOP_SEL := #Init,
               L_AUT := #Init,
               L_REMOTE := #Init,
               L_RESET := #Reset,
               L_MON := #Init,
               INSTANCE := 'AV-51.14');
END_REGION

REGION Network 17: AV-51.15
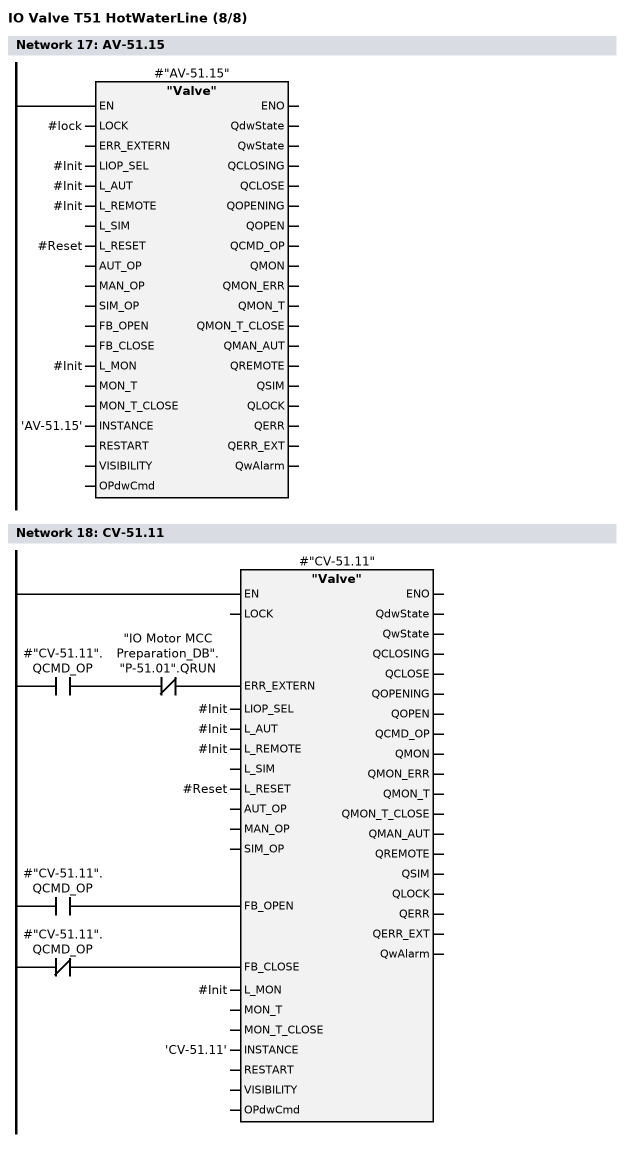
   RUNG wire#powerrail
      #"AV-51.15"(LOCK := #lock, ERR_EXTERN :=, LIOP_SEL := #Init, L_AUT := #Init, L_REMOTE := #Init, L_SIM :=, L_RESET := #Reset, AUT_OP :=, MAN_OP :=, SIM_OP :=, FB_OPEN :=, FB_CLOSE :=, L_MON := #Init, MON_T :=, MON_T_CLOSE :=, INSTANCE := 'AV-51.15', RESTART :=, VISIBILITY :=, OPdwCmd :=, QdwState =>, QwState =>, QCLOSING =>, QCLOSE =>, QOPENING =>, QOPEN =>, QCMD_OP =>, QMON =>, QMON_ERR =>, QMON_T =>, QMON_T_CLOSE =>, QMAN_AUT =>, QREMOTE =>, QSIM =>, QLOCK =>, QERR =>, QERR_EXT =>, QwAlarm =>)
   END_RUNG
   // the same network as SCL:
   #"AV-51.15"(LOCK := #lock,   // "Valve"
               LIOP_SEL := #Init,
               L_AUT := #Init,
               L_REMOTE := #Init,
               L_RESET := #Reset,
               L_MON := #Init,
               INSTANCE := 'AV-51.15');
END_REGION

REGION Network 18: CV-51.11
   RUNG wire#powerrail
      #"CV-51.11"(ERR_EXTERN := wire#w1, FB_OPEN := wire#w2, FB_CLOSE := wire#w3, LOCK :=, LIOP_SEL := #Init, L_AUT := #Init, L_REMOTE := #Init, L_SIM :=, L_RESET := #Reset, AUT_OP :=, MAN_OP :=, SIM_OP :=, L_MON := #Init, MON_T :=, MON_T_CLOSE :=, INSTANCE := 'CV-51.11', RESTART :=, VISIBILITY :=, OPdwCmd :=, QdwState =>, QwState =>, QCLOSING =>, QCLOSE =>, QOPENING =>, QOPEN =>, QCMD_OP =>, QMON =>, QMON_ERR =>, QMON_T =>, QMON_T_CLOSE =>, QMAN_AUT =>, QREMOTE =>, QSIM =>, QLOCK =>, QERR =>, QERR_EXT =>, QwAlarm =>)
   END_RUNG
   RUNG wire#powerrail
      Contact( #"CV-51.11".QCMD_OP )
      I_Contact( "IO Motor MCC Preparation_DB"."P-51.01".QRUN )
   END_RUNG wire#w1
   RUNG wire#powerrail
      Contact( #"CV-51.11".QCMD_OP )
   END_RUNG wire#w2
   RUNG wire#powerrail
      I_Contact( #"CV-51.11".QCMD_OP )
   END_RUNG wire#w3
   // the same network as SCL:
   #"CV-51.11"(ERR_EXTERN := #"CV-51.11".QCMD_OP AND NOT "IO Motor MCC Preparation_DB"."P-51.01".QRUN,   // "Valve"
               LIOP_SEL := #Init,
               L_AUT := #Init,
               L_REMOTE := #Init,
               L_RESET := #Reset,
               FB_OPEN := #"CV-51.11".QCMD_OP,
               FB_CLOSE := NOT #"CV-51.11".QCMD_OP,
               L_MON := #Init,
               INSTANCE := 'CV-51.11');
END_REGION
END_FUNCTION_BLOCK

FUNCTION "IO Homoge" : Void   // FC1, LAD
{ S7_Optimized_Access := 'TRUE' }
VERSION : 0.1
// stored: AutoNumber true, IsIECCheckEnabled false, SetENOAutomatically false, UDAEnableTagReadback false
BEGIN

REGION Network 1: Analog
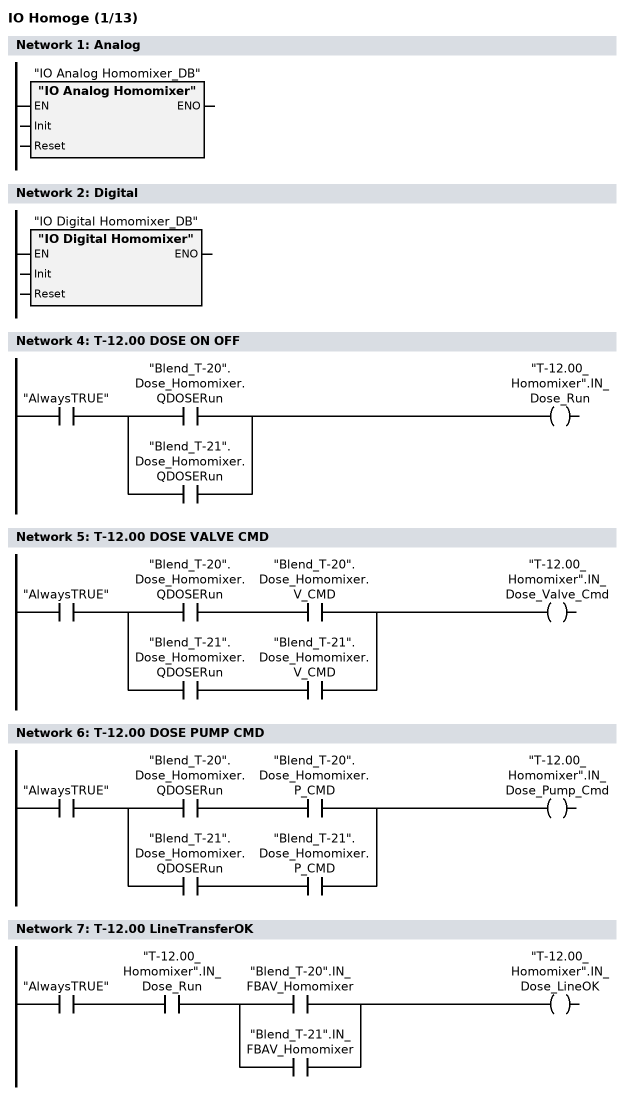
   RUNG wire#powerrail
      "IO Analog Homomixer_DB"(Init :=, Reset :=)
   END_RUNG
   // the same network as SCL:
   "IO Analog Homomixer_DB"();   // "IO Analog Homomixer"
END_REGION

REGION Network 2: Digital
   RUNG wire#powerrail
      "IO Digital Homomixer_DB"(Init :=, Reset :=)
   END_RUNG
   // the same network as SCL:
   "IO Digital Homomixer_DB"();   // "IO Digital Homomixer"
END_REGION

REGION Network 4: T-12.00 DOSE ON OFF
   RUNG wire#powerrail
      Contact( "AlwaysTRUE" )
      wire#w1
      Contact( "Blend_T-20".Dose_Homomixer.QDOSERun )
      wire#w2
      Coil( "T-12.00_Homomixer".IN_Dose_Run )
   END_RUNG
   RUNG wire#w1
      Contact( "Blend_T-21".Dose_Homomixer.QDOSERun )
   END_RUNG wire#w2
   // the same network as SCL:
   "T-12.00_Homomixer".IN_Dose_Run := "AlwaysTRUE" AND ("Blend_T-20".Dose_Homomixer.QDOSERun OR "Blend_T-21".Dose_Homomixer.QDOSERun);
END_REGION

REGION Network 5: T-12.00 DOSE VALVE CMD
   RUNG wire#powerrail
      Contact( "AlwaysTRUE" )
      wire#w1
      Contact( "Blend_T-20".Dose_Homomixer.QDOSERun )
      Contact( "Blend_T-20".Dose_Homomixer.V_CMD )
      wire#w2
      Coil( "T-12.00_Homomixer".IN_Dose_Valve_Cmd )
   END_RUNG
   RUNG wire#w1
      Contact( "Blend_T-21".Dose_Homomixer.QDOSERun )
      Contact( "Blend_T-21".Dose_Homomixer.V_CMD )
   END_RUNG wire#w2
   // the same network as SCL:
   "T-12.00_Homomixer".IN_Dose_Valve_Cmd := "AlwaysTRUE" AND (("Blend_T-20".Dose_Homomixer.QDOSERun AND "Blend_T-20".Dose_Homomixer.V_CMD) OR ("Blend_T-21".Dose_Homomixer.QDOSERun AND "Blend_T-21".Dose_Homomixer.V_CMD));
END_REGION

REGION Network 6: T-12.00 DOSE PUMP CMD
   RUNG wire#powerrail
      Contact( "AlwaysTRUE" )
      wire#w1
      Contact( "Blend_T-20".Dose_Homomixer.QDOSERun )
      Contact( "Blend_T-20".Dose_Homomixer.P_CMD )
      wire#w2
      Coil( "T-12.00_Homomixer".IN_Dose_Pump_Cmd )
   END_RUNG
   RUNG wire#w1
      Contact( "Blend_T-21".Dose_Homomixer.QDOSERun )
      Contact( "Blend_T-21".Dose_Homomixer.P_CMD )
   END_RUNG wire#w2
   // the same network as SCL:
   "T-12.00_Homomixer".IN_Dose_Pump_Cmd := "AlwaysTRUE" AND (("Blend_T-20".Dose_Homomixer.QDOSERun AND "Blend_T-20".Dose_Homomixer.P_CMD) OR ("Blend_T-21".Dose_Homomixer.QDOSERun AND "Blend_T-21".Dose_Homomixer.P_CMD));
END_REGION

REGION Network 7: T-12.00 LineTransferOK
   RUNG wire#powerrail
      Contact( "AlwaysTRUE" )
      Contact( "T-12.00_Homomixer".IN_Dose_Run )
      wire#w1
      Contact( "Blend_T-20".IN_FBAV_Homomixer )
      wire#w2
      Coil( "T-12.00_Homomixer".IN_Dose_LineOK )
   END_RUNG
   RUNG wire#w1
      Contact( "Blend_T-21".IN_FBAV_Homomixer )
   END_RUNG wire#w2
   // the same network as SCL:
   "T-12.00_Homomixer".IN_Dose_LineOK := "AlwaysTRUE" AND "T-12.00_Homomixer".IN_Dose_Run AND ("Blend_T-20".IN_FBAV_Homomixer OR "Blend_T-21".IN_FBAV_Homomixer);
END_REGION

REGION Network 8: T-12.00 Homomixer
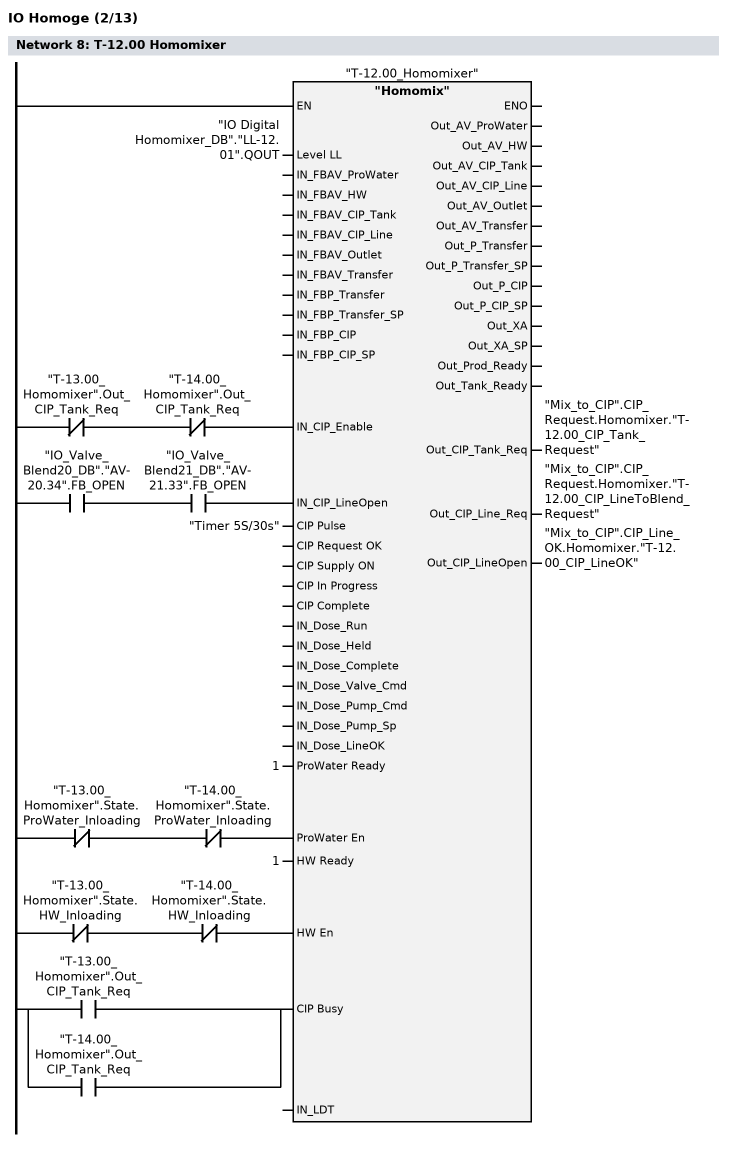
   RUNG wire#powerrail
      "T-12.00_Homomixer"(IN_CIP_Enable := wire#w1, IN_CIP_LineOpen := wire#w2, "ProWater En" := wire#w3, "HW En" := wire#w4, "CIP Busy" := wire#w5, "Level LL" := "IO Digital Homomixer_DB"."LL-12.01".QOUT, IN_FBAV_ProWater :=, IN_FBAV_HW :=, IN_FBAV_CIP_Tank :=, IN_FBAV_CIP_Line :=, IN_FBAV_Outlet :=, IN_FBAV_Transfer :=, IN_FBP_Transfer :=, IN_FBP_Transfer_SP :=, IN_FBP_CIP :=, IN_FBP_CIP_SP :=, "CIP Pulse" := "Timer 5S/30s", "CIP Request OK" :=, "CIP Supply ON" :=, "CIP In Progress" :=, "CIP Complete" :=, IN_Dose_Run :=, IN_Dose_Held :=, IN_Dose_Complete :=, IN_Dose_Valve_Cmd :=, IN_Dose_Pump_Cmd :=, IN_Dose_Pump_Sp :=, IN_Dose_LineOK :=, "ProWater Ready" := 1, "HW Ready" := 1, IN_LDT :=, Out_AV_ProWater =>, Out_AV_HW =>, Out_AV_CIP_Tank =>, Out_AV_CIP_Line =>, Out_AV_Outlet =>, Out_AV_Transfer =>, Out_P_Transfer =>, Out_P_Transfer_SP =>, Out_P_CIP =>, Out_P_CIP_SP =>, Out_XA =>, Out_XA_SP =>, Out_Prod_Ready =>, Out_Tank_Ready =>, Out_CIP_Tank_Req => "Mix_to_CIP".CIP_Request.Homomixer."T-12.00_CIP_Tank_Request", Out_CIP_Line_Req => "Mix_to_CIP".CIP_Request.Homomixer."T-12.00_CIP_LineToBlend_Request", Out_CIP_LineOpen => "Mix_to_CIP".CIP_Line_OK.Homomixer."T-12.00_CIP_LineOK")
   END_RUNG
   RUNG wire#powerrail
      I_Contact( "T-13.00_Homomixer".Out_CIP_Tank_Req )
      I_Contact( "T-14.00_Homomixer".Out_CIP_Tank_Req )
   END_RUNG wire#w1
   RUNG wire#powerrail
      Contact( "IO_Valve_Blend20_DB"."AV-20.34".FB_OPEN )
      Contact( "IO_Valve_Blend21_DB"."AV-21.33".FB_OPEN )
   END_RUNG wire#w2
   RUNG wire#powerrail
      I_Contact( "T-13.00_Homomixer".State.ProWater_Inloading )
      I_Contact( "T-14.00_Homomixer".State.ProWater_Inloading )
   END_RUNG wire#w3
   RUNG wire#powerrail
      I_Contact( "T-13.00_Homomixer".State.HW_Inloading )
      I_Contact( "T-14.00_Homomixer".State.HW_Inloading )
   END_RUNG wire#w4
   RUNG wire#powerrail
      Contact( "T-13.00_Homomixer".Out_CIP_Tank_Req )
   END_RUNG wire#w5
   RUNG wire#powerrail
      Contact( "T-14.00_Homomixer".Out_CIP_Tank_Req )
   END_RUNG wire#w5
   // the same network as SCL:
   "T-12.00_Homomixer"("Level LL" := "IO Digital Homomixer_DB"."LL-12.01".QOUT,   // "Homomix"
                       IN_CIP_Enable := NOT "T-13.00_Homomixer".Out_CIP_Tank_Req AND NOT "T-14.00_Homomixer".Out_CIP_Tank_Req,
                       IN_CIP_LineOpen := "IO_Valve_Blend20_DB"."AV-20.34".FB_OPEN AND "IO_Valve_Blend21_DB"."AV-21.33".FB_OPEN,
                       "CIP Pulse" := "Timer 5S/30s",
                       "ProWater Ready" := 1,
                       "ProWater En" := NOT "T-13.00_Homomixer".State.ProWater_Inloading AND NOT "T-14.00_Homomixer".State.ProWater_Inloading,
                       "HW Ready" := 1,
                       "HW En" := NOT "T-13.00_Homomixer".State.HW_Inloading AND NOT "T-14.00_Homomixer".State.HW_Inloading,
                       "CIP Busy" := "T-13.00_Homomixer".Out_CIP_Tank_Req OR "T-14.00_Homomixer".Out_CIP_Tank_Req,
                       Out_CIP_Tank_Req => "Mix_to_CIP".CIP_Request.Homomixer."T-12.00_CIP_Tank_Request",
                       Out_CIP_Line_Req => "Mix_to_CIP".CIP_Request.Homomixer."T-12.00_CIP_LineToBlend_Request",
                       Out_CIP_LineOpen => "Mix_to_CIP".CIP_Line_OK.Homomixer."T-12.00_CIP_LineOK");
END_REGION

REGION Network 9: T-12.00 Valve Cmd
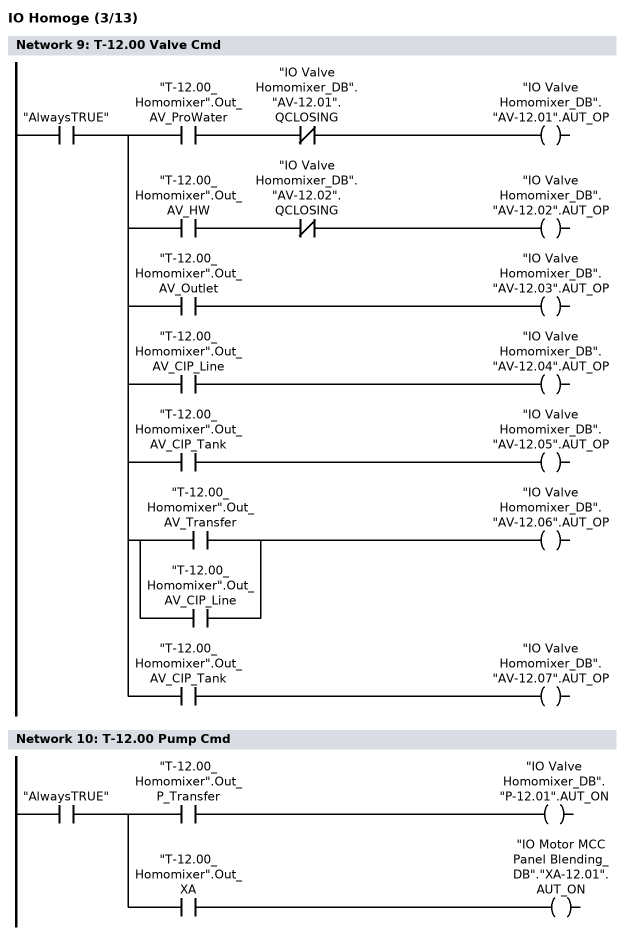
   RUNG wire#powerrail
      Contact( "AlwaysTRUE" )
      wire#w1
      Contact( "T-12.00_Homomixer".Out_AV_ProWater )
      I_Contact( "IO Valve Homomixer_DB"."AV-12.01".QCLOSING )
      Coil( "IO Valve Homomixer_DB"."AV-12.01".AUT_OP )
   END_RUNG
   RUNG wire#w1
      Contact( "T-12.00_Homomixer".Out_AV_HW )
      I_Contact( "IO Valve Homomixer_DB"."AV-12.02".QCLOSING )
      Coil( "IO Valve Homomixer_DB"."AV-12.02".AUT_OP )
   END_RUNG
   RUNG wire#w1
      Contact( "T-12.00_Homomixer".Out_AV_Outlet )
      Coil( "IO Valve Homomixer_DB"."AV-12.03".AUT_OP )
   END_RUNG
   RUNG wire#w1
      Contact( "T-12.00_Homomixer".Out_AV_CIP_Line )
      Coil( "IO Valve Homomixer_DB"."AV-12.04".AUT_OP )
   END_RUNG
   RUNG wire#w1
      Contact( "T-12.00_Homomixer".Out_AV_CIP_Tank )
      Coil( "IO Valve Homomixer_DB"."AV-12.05".AUT_OP )
   END_RUNG
   RUNG wire#w1
      Contact( "T-12.00_Homomixer".Out_AV_Transfer )
      wire#w2
      Coil( "IO Valve Homomixer_DB"."AV-12.06".AUT_OP )
   END_RUNG
   RUNG wire#w1
      Contact( "T-12.00_Homomixer".Out_AV_CIP_Line )
   END_RUNG wire#w2
   RUNG wire#w1
      Contact( "T-12.00_Homomixer".Out_AV_CIP_Tank )
      Coil( "IO Valve Homomixer_DB"."AV-12.07".AUT_OP )
   END_RUNG
   // the same network as SCL:
   "IO Valve Homomixer_DB"."AV-12.01".AUT_OP := "AlwaysTRUE" AND "T-12.00_Homomixer".Out_AV_ProWater AND NOT "IO Valve Homomixer_DB"."AV-12.01".QCLOSING;
   "IO Valve Homomixer_DB"."AV-12.02".AUT_OP := "AlwaysTRUE" AND "T-12.00_Homomixer".Out_AV_HW AND NOT "IO Valve Homomixer_DB"."AV-12.02".QCLOSING;
   "IO Valve Homomixer_DB"."AV-12.03".AUT_OP := "AlwaysTRUE" AND "T-12.00_Homomixer".Out_AV_Outlet;
   "IO Valve Homomixer_DB"."AV-12.04".AUT_OP := "AlwaysTRUE" AND "T-12.00_Homomixer".Out_AV_CIP_Line;
   "IO Valve Homomixer_DB"."AV-12.05".AUT_OP := "AlwaysTRUE" AND "T-12.00_Homomixer".Out_AV_CIP_Tank;
   "IO Valve Homomixer_DB"."AV-12.06".AUT_OP := "AlwaysTRUE" AND ("T-12.00_Homomixer".Out_AV_Transfer OR "T-12.00_Homomixer".Out_AV_CIP_Line);
   "IO Valve Homomixer_DB"."AV-12.07".AUT_OP := "AlwaysTRUE" AND "T-12.00_Homomixer".Out_AV_CIP_Tank;
END_REGION

REGION Network 10: T-12.00 Pump Cmd
   RUNG wire#powerrail
      Contact( "AlwaysTRUE" )
      wire#w1
      Contact( "T-12.00_Homomixer".Out_P_Transfer )
      Coil( "IO Valve Homomixer_DB"."P-12.01".AUT_ON )
   END_RUNG
   RUNG wire#w1
      Contact( "T-12.00_Homomixer".Out_XA )
      Coil( "IO Motor MCC Panel Blending_DB"."XA-12.01".AUT_ON )
   END_RUNG
   // the same network as SCL:
   "IO Valve Homomixer_DB"."P-12.01".AUT_ON := "AlwaysTRUE" AND "T-12.00_Homomixer".Out_P_Transfer;
   "IO Motor MCC Panel Blending_DB"."XA-12.01".AUT_ON := "AlwaysTRUE" AND "T-12.00_Homomixer".Out_XA;
END_REGION

REGION Network 11: T-12.00 Feedback Instrument
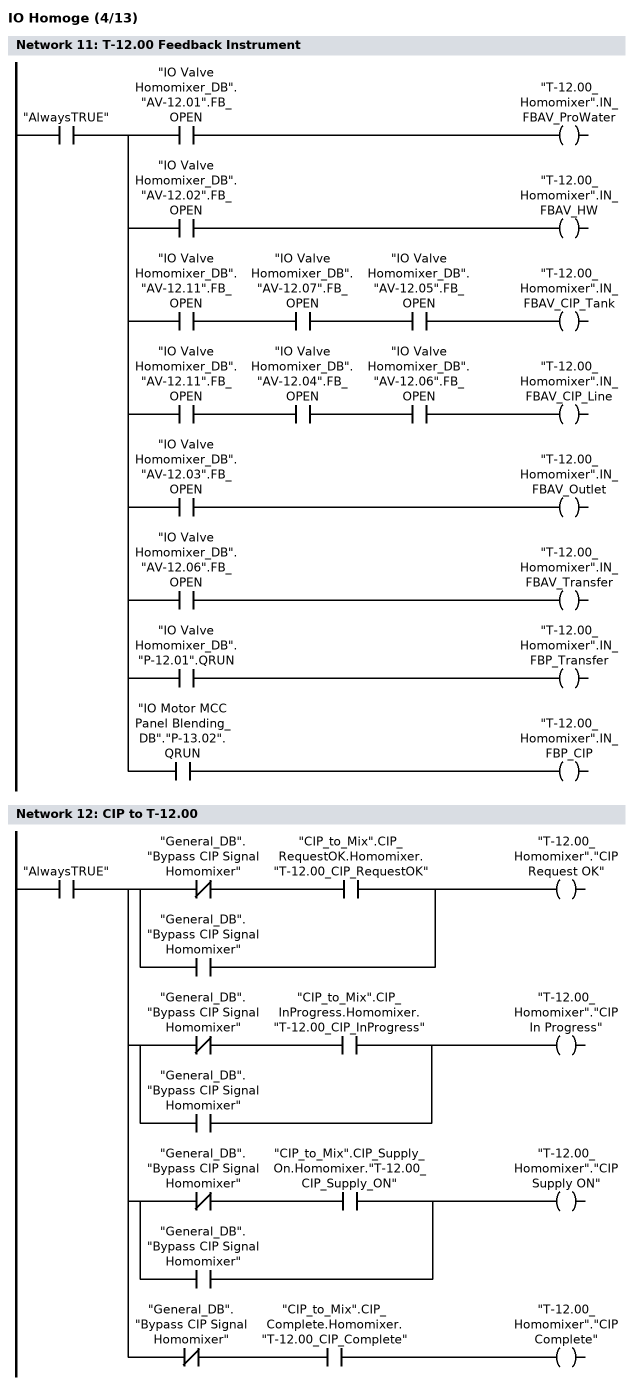
   RUNG wire#powerrail
      Contact( "AlwaysTRUE" )
      wire#w1
      Contact( "IO Valve Homomixer_DB"."AV-12.01".FB_OPEN )
      Coil( "T-12.00_Homomixer".IN_FBAV_ProWater )
   END_RUNG
   RUNG wire#w1
      Contact( "IO Valve Homomixer_DB"."AV-12.02".FB_OPEN )
      Coil( "T-12.00_Homomixer".IN_FBAV_HW )
   END_RUNG
   RUNG wire#w1
      Contact( "IO Valve Homomixer_DB"."AV-12.11".FB_OPEN )
      Contact( "IO Valve Homomixer_DB"."AV-12.07".FB_OPEN )
      Contact( "IO Valve Homomixer_DB"."AV-12.05".FB_OPEN )
      Coil( "T-12.00_Homomixer".IN_FBAV_CIP_Tank )
   END_RUNG
   RUNG wire#w1
      Contact( "IO Valve Homomixer_DB"."AV-12.11".FB_OPEN )
      Contact( "IO Valve Homomixer_DB"."AV-12.04".FB_OPEN )
      Contact( "IO Valve Homomixer_DB"."AV-12.06".FB_OPEN )
      Coil( "T-12.00_Homomixer".IN_FBAV_CIP_Line )
   END_RUNG
   RUNG wire#w1
      Contact( "IO Valve Homomixer_DB"."AV-12.03".FB_OPEN )
      Coil( "T-12.00_Homomixer".IN_FBAV_Outlet )
   END_RUNG
   RUNG wire#w1
      Contact( "IO Valve Homomixer_DB"."AV-12.06".FB_OPEN )
      Coil( "T-12.00_Homomixer".IN_FBAV_Transfer )
   END_RUNG
   RUNG wire#w1
      Contact( "IO Valve Homomixer_DB"."P-12.01".QRUN )
      Coil( "T-12.00_Homomixer".IN_FBP_Transfer )
   END_RUNG
   RUNG wire#w1
      Contact( "IO Motor MCC Panel Blending_DB"."P-13.02".QRUN )
      Coil( "T-12.00_Homomixer".IN_FBP_CIP )
   END_RUNG
   // the same network as SCL:
   "T-12.00_Homomixer".IN_FBAV_ProWater := "AlwaysTRUE" AND "IO Valve Homomixer_DB"."AV-12.01".FB_OPEN;
   "T-12.00_Homomixer".IN_FBAV_HW := "AlwaysTRUE" AND "IO Valve Homomixer_DB"."AV-12.02".FB_OPEN;
   "T-12.00_Homomixer".IN_FBAV_CIP_Tank := "AlwaysTRUE" AND "IO Valve Homomixer_DB"."AV-12.11".FB_OPEN AND "IO Valve Homomixer_DB"."AV-12.07".FB_OPEN AND "IO Valve Homomixer_DB"."AV-12.05".FB_OPEN;
   "T-12.00_Homomixer".IN_FBAV_CIP_Line := "AlwaysTRUE" AND "IO Valve Homomixer_DB"."AV-12.11".FB_OPEN AND "IO Valve Homomixer_DB"."AV-12.04".FB_OPEN AND "IO Valve Homomixer_DB"."AV-12.06".FB_OPEN;
   "T-12.00_Homomixer".IN_FBAV_Outlet := "AlwaysTRUE" AND "IO Valve Homomixer_DB"."AV-12.03".FB_OPEN;
   "T-12.00_Homomixer".IN_FBAV_Transfer := "AlwaysTRUE" AND "IO Valve Homomixer_DB"."AV-12.06".FB_OPEN;
   "T-12.00_Homomixer".IN_FBP_Transfer := "AlwaysTRUE" AND "IO Valve Homomixer_DB"."P-12.01".QRUN;
   "T-12.00_Homomixer".IN_FBP_CIP := "AlwaysTRUE" AND "IO Motor MCC Panel Blending_DB"."P-13.02".QRUN;
END_REGION

REGION Network 12: CIP to T-12.00
   RUNG wire#powerrail
      Contact( "AlwaysTRUE" )
      wire#w1
      I_Contact( "General_DB"."Bypass CIP Signal Homomixer" )
      Contact( "CIP_to_Mix".CIP_RequestOK.Homomixer."T-12.00_CIP_RequestOK" )
      wire#w2
      Coil( "T-12.00_Homomixer"."CIP Request OK" )
   END_RUNG
   RUNG wire#w1
      Contact( "General_DB"."Bypass CIP Signal Homomixer" )
   END_RUNG wire#w2
   RUNG wire#w1
      I_Contact( "General_DB"."Bypass CIP Signal Homomixer" )
      Contact( "CIP_to_Mix".CIP_InProgress.Homomixer."T-12.00_CIP_InProgress" )
      wire#w3
      Coil( "T-12.00_Homomixer"."CIP In Progress" )
   END_RUNG
   RUNG wire#w1
      Contact( "General_DB"."Bypass CIP Signal Homomixer" )
   END_RUNG wire#w3
   RUNG wire#w1
      I_Contact( "General_DB"."Bypass CIP Signal Homomixer" )
      Contact( "CIP_to_Mix".CIP_Supply_On.Homomixer."T-12.00_CIP_Supply_ON" )
      wire#w4
      Coil( "T-12.00_Homomixer"."CIP Supply ON" )
   END_RUNG
   RUNG wire#w1
      Contact( "General_DB"."Bypass CIP Signal Homomixer" )
   END_RUNG wire#w4
   RUNG wire#w1
      I_Contact( "General_DB"."Bypass CIP Signal Homomixer" )
      Contact( "CIP_to_Mix".CIP_Complete.Homomixer."T-12.00_CIP_Complete" )
      Coil( "T-12.00_Homomixer"."CIP Complete" )
   END_RUNG
   // the same network as SCL:
   "T-12.00_Homomixer"."CIP Request OK" := "AlwaysTRUE" AND ((NOT "General_DB"."Bypass CIP Signal Homomixer" AND "CIP_to_Mix".CIP_RequestOK.Homomixer."T-12.00_CIP_RequestOK") OR "General_DB"."Bypass CIP Signal Homomixer");
   "T-12.00_Homomixer"."CIP In Progress" := "AlwaysTRUE" AND ((NOT "General_DB"."Bypass CIP Signal Homomixer" AND "CIP_to_Mix".CIP_InProgress.Homomixer."T-12.00_CIP_InProgress") OR "General_DB"."Bypass CIP Signal Homomixer");
   "T-12.00_Homomixer"."CIP Supply ON" := "AlwaysTRUE" AND ((NOT "General_DB"."Bypass CIP Signal Homomixer" AND "CIP_to_Mix".CIP_Supply_On.Homomixer."T-12.00_CIP_Supply_ON") OR "General_DB"."Bypass CIP Signal Homomixer");
   "T-12.00_Homomixer"."CIP Complete" := "AlwaysTRUE" AND NOT "General_DB"."Bypass CIP Signal Homomixer" AND "CIP_to_Mix".CIP_Complete.Homomixer."T-12.00_CIP_Complete";
END_REGION

REGION Network 15: T-13.00 DOSE ON OFF
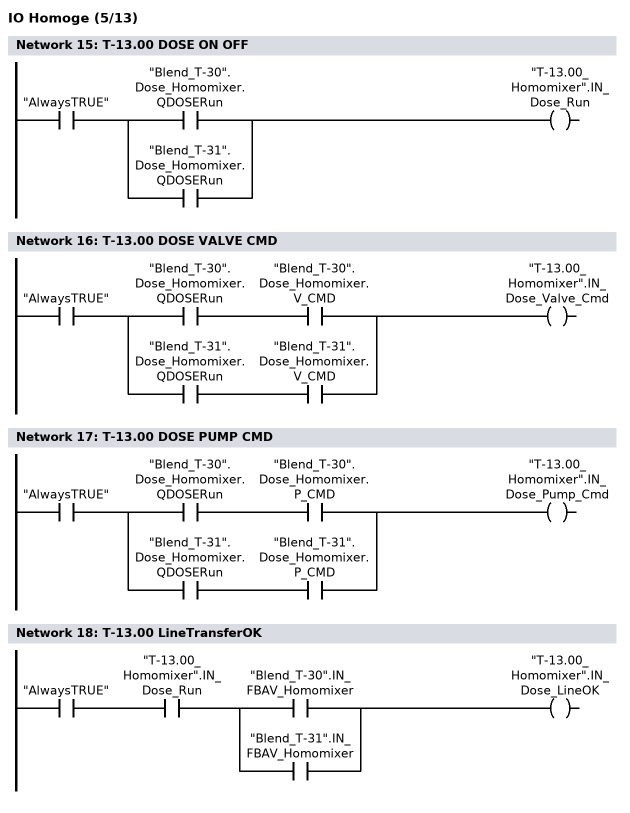
   RUNG wire#powerrail
      Contact( "AlwaysTRUE" )
      wire#w1
      Contact( "Blend_T-30".Dose_Homomixer.QDOSERun )
      wire#w2
      Coil( "T-13.00_Homomixer".IN_Dose_Run )
   END_RUNG
   RUNG wire#w1
      Contact( "Blend_T-31".Dose_Homomixer.QDOSERun )
   END_RUNG wire#w2
   // the same network as SCL:
   "T-13.00_Homomixer".IN_Dose_Run := "AlwaysTRUE" AND ("Blend_T-30".Dose_Homomixer.QDOSERun OR "Blend_T-31".Dose_Homomixer.QDOSERun);
END_REGION

REGION Network 16: T-13.00 DOSE VALVE CMD
   RUNG wire#powerrail
      Contact( "AlwaysTRUE" )
      wire#w1
      Contact( "Blend_T-30".Dose_Homomixer.QDOSERun )
      Contact( "Blend_T-30".Dose_Homomixer.V_CMD )
      wire#w2
      Coil( "T-13.00_Homomixer".IN_Dose_Valve_Cmd )
   END_RUNG
   RUNG wire#w1
      Contact( "Blend_T-31".Dose_Homomixer.QDOSERun )
      Contact( "Blend_T-31".Dose_Homomixer.V_CMD )
   END_RUNG wire#w2
   // the same network as SCL:
   "T-13.00_Homomixer".IN_Dose_Valve_Cmd := "AlwaysTRUE" AND (("Blend_T-30".Dose_Homomixer.QDOSERun AND "Blend_T-30".Dose_Homomixer.V_CMD) OR ("Blend_T-31".Dose_Homomixer.QDOSERun AND "Blend_T-31".Dose_Homomixer.V_CMD));
END_REGION

REGION Network 17: T-13.00 DOSE PUMP CMD
   RUNG wire#powerrail
      Contact( "AlwaysTRUE" )
      wire#w1
      Contact( "Blend_T-30".Dose_Homomixer.QDOSERun )
      Contact( "Blend_T-30".Dose_Homomixer.P_CMD )
      wire#w2
      Coil( "T-13.00_Homomixer".IN_Dose_Pump_Cmd )
   END_RUNG
   RUNG wire#w1
      Contact( "Blend_T-31".Dose_Homomixer.QDOSERun )
      Contact( "Blend_T-31".Dose_Homomixer.P_CMD )
   END_RUNG wire#w2
   // the same network as SCL:
   "T-13.00_Homomixer".IN_Dose_Pump_Cmd := "AlwaysTRUE" AND (("Blend_T-30".Dose_Homomixer.QDOSERun AND "Blend_T-30".Dose_Homomixer.P_CMD) OR ("Blend_T-31".Dose_Homomixer.QDOSERun AND "Blend_T-31".Dose_Homomixer.P_CMD));
END_REGION

REGION Network 18: T-13.00 LineTransferOK
   RUNG wire#powerrail
      Contact( "AlwaysTRUE" )
      Contact( "T-13.00_Homomixer".IN_Dose_Run )
      wire#w1
      Contact( "Blend_T-30".IN_FBAV_Homomixer )
      wire#w2
      Coil( "T-13.00_Homomixer".IN_Dose_LineOK )
   END_RUNG
   RUNG wire#w1
      Contact( "Blend_T-31".IN_FBAV_Homomixer )
   END_RUNG wire#w2
   // the same network as SCL:
   "T-13.00_Homomixer".IN_Dose_LineOK := "AlwaysTRUE" AND "T-13.00_Homomixer".IN_Dose_Run AND ("Blend_T-30".IN_FBAV_Homomixer OR "Blend_T-31".IN_FBAV_Homomixer);
END_REGION

REGION Network 19: T-13.00 Homomixer
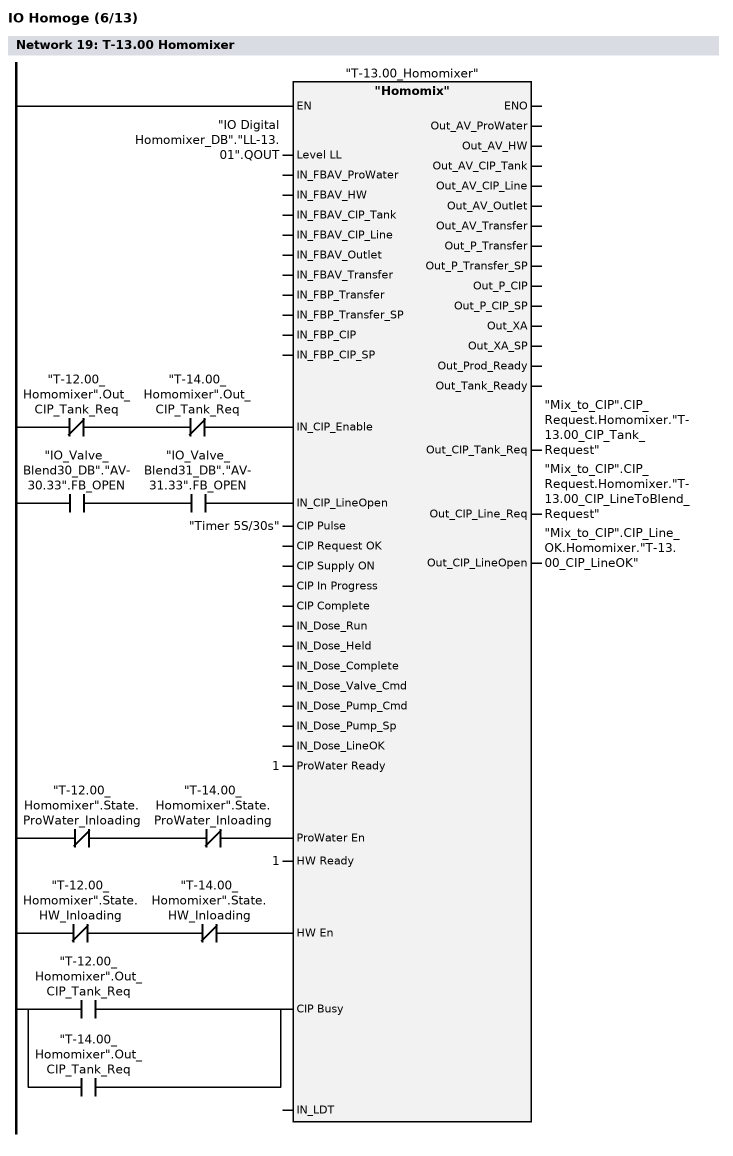
   RUNG wire#powerrail
      "T-13.00_Homomixer"(IN_CIP_Enable := wire#w1, IN_CIP_LineOpen := wire#w2, "ProWater En" := wire#w3, "HW En" := wire#w4, "CIP Busy" := wire#w5, "Level LL" := "IO Digital Homomixer_DB"."LL-13.01".QOUT, IN_FBAV_ProWater :=, IN_FBAV_HW :=, IN_FBAV_CIP_Tank :=, IN_FBAV_CIP_Line :=, IN_FBAV_Outlet :=, IN_FBAV_Transfer :=, IN_FBP_Transfer :=, IN_FBP_Transfer_SP :=, IN_FBP_CIP :=, IN_FBP_CIP_SP :=, "CIP Pulse" := "Timer 5S/30s", "CIP Request OK" :=, "CIP Supply ON" :=, "CIP In Progress" :=, "CIP Complete" :=, IN_Dose_Run :=, IN_Dose_Held :=, IN_Dose_Complete :=, IN_Dose_Valve_Cmd :=, IN_Dose_Pump_Cmd :=, IN_Dose_Pump_Sp :=, IN_Dose_LineOK :=, "ProWater Ready" := 1, "HW Ready" := 1, IN_LDT :=, Out_AV_ProWater =>, Out_AV_HW =>, Out_AV_CIP_Tank =>, Out_AV_CIP_Line =>, Out_AV_Outlet =>, Out_AV_Transfer =>, Out_P_Transfer =>, Out_P_Transfer_SP =>, Out_P_CIP =>, Out_P_CIP_SP =>, Out_XA =>, Out_XA_SP =>, Out_Prod_Ready =>, Out_Tank_Ready =>, Out_CIP_Tank_Req => "Mix_to_CIP".CIP_Request.Homomixer."T-13.00_CIP_Tank_Request", Out_CIP_Line_Req => "Mix_to_CIP".CIP_Request.Homomixer."T-13.00_CIP_LineToBlend_Request", Out_CIP_LineOpen => "Mix_to_CIP".CIP_Line_OK.Homomixer."T-13.00_CIP_LineOK")
   END_RUNG
   RUNG wire#powerrail
      I_Contact( "T-12.00_Homomixer".Out_CIP_Tank_Req )
      I_Contact( "T-14.00_Homomixer".Out_CIP_Tank_Req )
   END_RUNG wire#w1
   RUNG wire#powerrail
      Contact( "IO_Valve_Blend30_DB"."AV-30.33".FB_OPEN )
      Contact( "IO_Valve_Blend31_DB"."AV-31.33".FB_OPEN )
   END_RUNG wire#w2
   RUNG wire#powerrail
      I_Contact( "T-12.00_Homomixer".State.ProWater_Inloading )
      I_Contact( "T-14.00_Homomixer".State.ProWater_Inloading )
   END_RUNG wire#w3
   RUNG wire#powerrail
      I_Contact( "T-12.00_Homomixer".State.HW_Inloading )
      I_Contact( "T-14.00_Homomixer".State.HW_Inloading )
   END_RUNG wire#w4
   RUNG wire#powerrail
      Contact( "T-12.00_Homomixer".Out_CIP_Tank_Req )
   END_RUNG wire#w5
   RUNG wire#powerrail
      Contact( "T-14.00_Homomixer".Out_CIP_Tank_Req )
   END_RUNG wire#w5
   // the same network as SCL:
   "T-13.00_Homomixer"("Level LL" := "IO Digital Homomixer_DB"."LL-13.01".QOUT,   // "Homomix"
                       IN_CIP_Enable := NOT "T-12.00_Homomixer".Out_CIP_Tank_Req AND NOT "T-14.00_Homomixer".Out_CIP_Tank_Req,
                       IN_CIP_LineOpen := "IO_Valve_Blend30_DB"."AV-30.33".FB_OPEN AND "IO_Valve_Blend31_DB"."AV-31.33".FB_OPEN,
                       "CIP Pulse" := "Timer 5S/30s",
                       "ProWater Ready" := 1,
                       "ProWater En" := NOT "T-12.00_Homomixer".State.ProWater_Inloading AND NOT "T-14.00_Homomixer".State.ProWater_Inloading,
                       "HW Ready" := 1,
                       "HW En" := NOT "T-12.00_Homomixer".State.HW_Inloading AND NOT "T-14.00_Homomixer".State.HW_Inloading,
                       "CIP Busy" := "T-12.00_Homomixer".Out_CIP_Tank_Req OR "T-14.00_Homomixer".Out_CIP_Tank_Req,
                       Out_CIP_Tank_Req => "Mix_to_CIP".CIP_Request.Homomixer."T-13.00_CIP_Tank_Request",
                       Out_CIP_Line_Req => "Mix_to_CIP".CIP_Request.Homomixer."T-13.00_CIP_LineToBlend_Request",
                       Out_CIP_LineOpen => "Mix_to_CIP".CIP_Line_OK.Homomixer."T-13.00_CIP_LineOK");
END_REGION

REGION Network 20: T-13.00 Valve Cmd
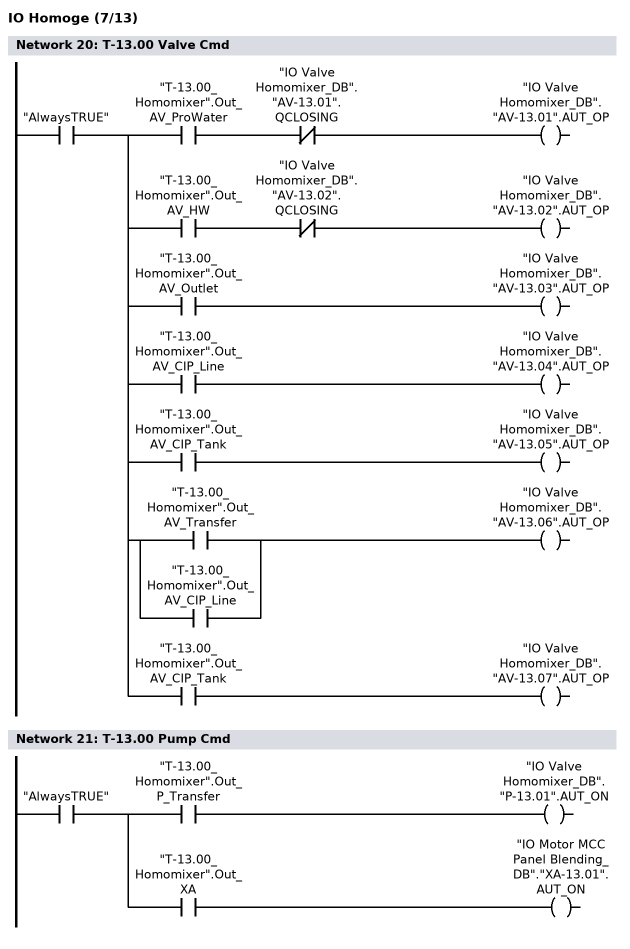
   RUNG wire#powerrail
      Contact( "AlwaysTRUE" )
      wire#w1
      Contact( "T-13.00_Homomixer".Out_AV_ProWater )
      I_Contact( "IO Valve Homomixer_DB"."AV-13.01".QCLOSING )
      Coil( "IO Valve Homomixer_DB"."AV-13.01".AUT_OP )
   END_RUNG
   RUNG wire#w1
      Contact( "T-13.00_Homomixer".Out_AV_HW )
      I_Contact( "IO Valve Homomixer_DB"."AV-13.02".QCLOSING )
      Coil( "IO Valve Homomixer_DB"."AV-13.02".AUT_OP )
   END_RUNG
   RUNG wire#w1
      Contact( "T-13.00_Homomixer".Out_AV_Outlet )
      Coil( "IO Valve Homomixer_DB"."AV-13.03".AUT_OP )
   END_RUNG
   RUNG wire#w1
      Contact( "T-13.00_Homomixer".Out_AV_CIP_Line )
      Coil( "IO Valve Homomixer_DB"."AV-13.04".AUT_OP )
   END_RUNG
   RUNG wire#w1
      Contact( "T-13.00_Homomixer".Out_AV_CIP_Tank )
      Coil( "IO Valve Homomixer_DB"."AV-13.05".AUT_OP )
   END_RUNG
   RUNG wire#w1
      Contact( "T-13.00_Homomixer".Out_AV_Transfer )
      wire#w2
      Coil( "IO Valve Homomixer_DB"."AV-13.06".AUT_OP )
   END_RUNG
   RUNG wire#w1
      Contact( "T-13.00_Homomixer".Out_AV_CIP_Line )
   END_RUNG wire#w2
   RUNG wire#w1
      Contact( "T-13.00_Homomixer".Out_AV_CIP_Tank )
      Coil( "IO Valve Homomixer_DB"."AV-13.07".AUT_OP )
   END_RUNG
   // the same network as SCL:
   "IO Valve Homomixer_DB"."AV-13.01".AUT_OP := "AlwaysTRUE" AND "T-13.00_Homomixer".Out_AV_ProWater AND NOT "IO Valve Homomixer_DB"."AV-13.01".QCLOSING;
   "IO Valve Homomixer_DB"."AV-13.02".AUT_OP := "AlwaysTRUE" AND "T-13.00_Homomixer".Out_AV_HW AND NOT "IO Valve Homomixer_DB"."AV-13.02".QCLOSING;
   "IO Valve Homomixer_DB"."AV-13.03".AUT_OP := "AlwaysTRUE" AND "T-13.00_Homomixer".Out_AV_Outlet;
   "IO Valve Homomixer_DB"."AV-13.04".AUT_OP := "AlwaysTRUE" AND "T-13.00_Homomixer".Out_AV_CIP_Line;
   "IO Valve Homomixer_DB"."AV-13.05".AUT_OP := "AlwaysTRUE" AND "T-13.00_Homomixer".Out_AV_CIP_Tank;
   "IO Valve Homomixer_DB"."AV-13.06".AUT_OP := "AlwaysTRUE" AND ("T-13.00_Homomixer".Out_AV_Transfer OR "T-13.00_Homomixer".Out_AV_CIP_Line);
   "IO Valve Homomixer_DB"."AV-13.07".AUT_OP := "AlwaysTRUE" AND "T-13.00_Homomixer".Out_AV_CIP_Tank;
END_REGION

REGION Network 21: T-13.00 Pump Cmd
   RUNG wire#powerrail
      Contact( "AlwaysTRUE" )
      wire#w1
      Contact( "T-13.00_Homomixer".Out_P_Transfer )
      Coil( "IO Valve Homomixer_DB"."P-13.01".AUT_ON )
   END_RUNG
   RUNG wire#w1
      Contact( "T-13.00_Homomixer".Out_XA )
      Coil( "IO Motor MCC Panel Blending_DB"."XA-13.01".AUT_ON )
   END_RUNG
   // the same network as SCL:
   "IO Valve Homomixer_DB"."P-13.01".AUT_ON := "AlwaysTRUE" AND "T-13.00_Homomixer".Out_P_Transfer;
   "IO Motor MCC Panel Blending_DB"."XA-13.01".AUT_ON := "AlwaysTRUE" AND "T-13.00_Homomixer".Out_XA;
END_REGION

REGION Network 22: T-13.00 Feedback Instrument
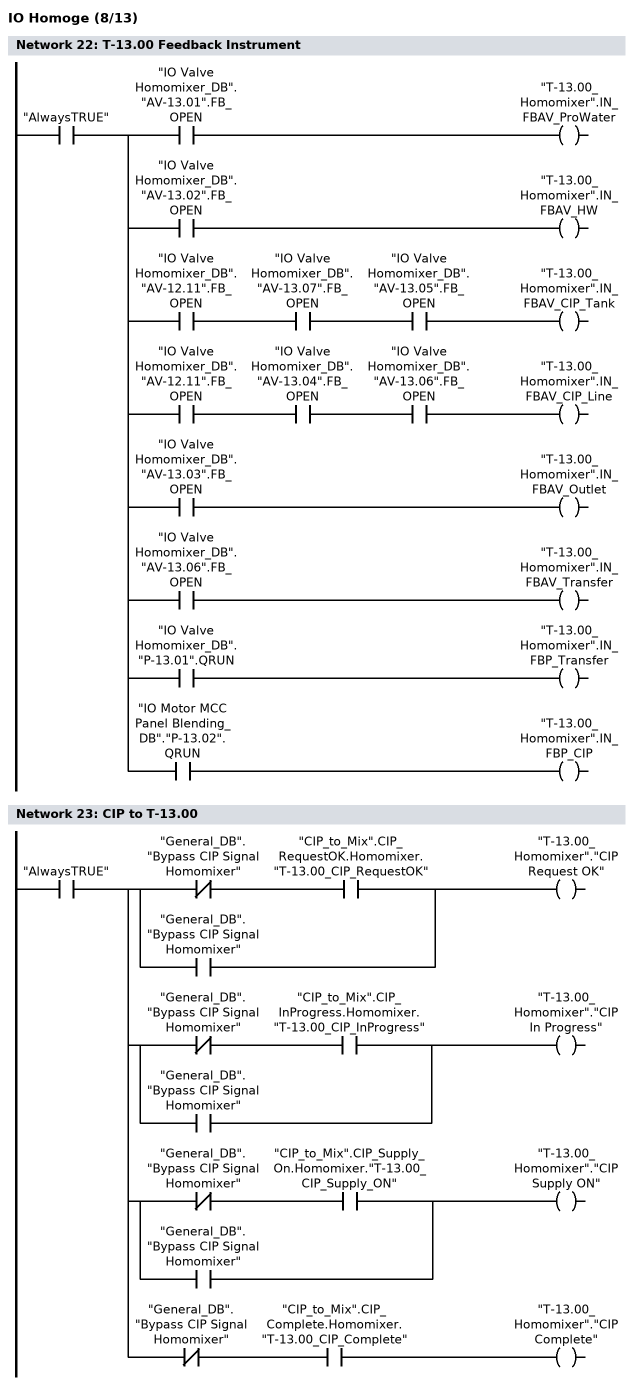
   RUNG wire#powerrail
      Contact( "AlwaysTRUE" )
      wire#w1
      Contact( "IO Valve Homomixer_DB"."AV-13.01".FB_OPEN )
      Coil( "T-13.00_Homomixer".IN_FBAV_ProWater )
   END_RUNG
   RUNG wire#w1
      Contact( "IO Valve Homomixer_DB"."AV-13.02".FB_OPEN )
      Coil( "T-13.00_Homomixer".IN_FBAV_HW )
   END_RUNG
   RUNG wire#w1
      Contact( "IO Valve Homomixer_DB"."AV-12.11".FB_OPEN )
      Contact( "IO Valve Homomixer_DB"."AV-13.07".FB_OPEN )
      Contact( "IO Valve Homomixer_DB"."AV-13.05".FB_OPEN )
      Coil( "T-13.00_Homomixer".IN_FBAV_CIP_Tank )
   END_RUNG
   RUNG wire#w1
      Contact( "IO Valve Homomixer_DB"."AV-12.11".FB_OPEN )
      Contact( "IO Valve Homomixer_DB"."AV-13.04".FB_OPEN )
      Contact( "IO Valve Homomixer_DB"."AV-13.06".FB_OPEN )
      Coil( "T-13.00_Homomixer".IN_FBAV_CIP_Line )
   END_RUNG
   RUNG wire#w1
      Contact( "IO Valve Homomixer_DB"."AV-13.03".FB_OPEN )
      Coil( "T-13.00_Homomixer".IN_FBAV_Outlet )
   END_RUNG
   RUNG wire#w1
      Contact( "IO Valve Homomixer_DB"."AV-13.06".FB_OPEN )
      Coil( "T-13.00_Homomixer".IN_FBAV_Transfer )
   END_RUNG
   RUNG wire#w1
      Contact( "IO Valve Homomixer_DB"."P-13.01".QRUN )
      Coil( "T-13.00_Homomixer".IN_FBP_Transfer )
   END_RUNG
   RUNG wire#w1
      Contact( "IO Motor MCC Panel Blending_DB"."P-13.02".QRUN )
      Coil( "T-13.00_Homomixer".IN_FBP_CIP )
   END_RUNG
   // the same network as SCL:
   "T-13.00_Homomixer".IN_FBAV_ProWater := "AlwaysTRUE" AND "IO Valve Homomixer_DB"."AV-13.01".FB_OPEN;
   "T-13.00_Homomixer".IN_FBAV_HW := "AlwaysTRUE" AND "IO Valve Homomixer_DB"."AV-13.02".FB_OPEN;
   "T-13.00_Homomixer".IN_FBAV_CIP_Tank := "AlwaysTRUE" AND "IO Valve Homomixer_DB"."AV-12.11".FB_OPEN AND "IO Valve Homomixer_DB"."AV-13.07".FB_OPEN AND "IO Valve Homomixer_DB"."AV-13.05".FB_OPEN;
   "T-13.00_Homomixer".IN_FBAV_CIP_Line := "AlwaysTRUE" AND "IO Valve Homomixer_DB"."AV-12.11".FB_OPEN AND "IO Valve Homomixer_DB"."AV-13.04".FB_OPEN AND "IO Valve Homomixer_DB"."AV-13.06".FB_OPEN;
   "T-13.00_Homomixer".IN_FBAV_Outlet := "AlwaysTRUE" AND "IO Valve Homomixer_DB"."AV-13.03".FB_OPEN;
   "T-13.00_Homomixer".IN_FBAV_Transfer := "AlwaysTRUE" AND "IO Valve Homomixer_DB"."AV-13.06".FB_OPEN;
   "T-13.00_Homomixer".IN_FBP_Transfer := "AlwaysTRUE" AND "IO Valve Homomixer_DB"."P-13.01".QRUN;
   "T-13.00_Homomixer".IN_FBP_CIP := "AlwaysTRUE" AND "IO Motor MCC Panel Blending_DB"."P-13.02".QRUN;
END_REGION

REGION Network 23: CIP to T-13.00
   RUNG wire#powerrail
      Contact( "AlwaysTRUE" )
      wire#w1
      I_Contact( "General_DB"."Bypass CIP Signal Homomixer" )
      Contact( "CIP_to_Mix".CIP_RequestOK.Homomixer."T-13.00_CIP_RequestOK" )
      wire#w2
      Coil( "T-13.00_Homomixer"."CIP Request OK" )
   END_RUNG
   RUNG wire#w1
      Contact( "General_DB"."Bypass CIP Signal Homomixer" )
   END_RUNG wire#w2
   RUNG wire#w1
      I_Contact( "General_DB"."Bypass CIP Signal Homomixer" )
      Contact( "CIP_to_Mix".CIP_InProgress.Homomixer."T-13.00_CIP_InProgress" )
      wire#w3
      Coil( "T-13.00_Homomixer"."CIP In Progress" )
   END_RUNG
   RUNG wire#w1
      Contact( "General_DB"."Bypass CIP Signal Homomixer" )
   END_RUNG wire#w3
   RUNG wire#w1
      I_Contact( "General_DB"."Bypass CIP Signal Homomixer" )
      Contact( "CIP_to_Mix".CIP_Supply_On.Homomixer."T-13.00_CIP_Supply_ON" )
      wire#w4
      Coil( "T-13.00_Homomixer"."CIP Supply ON" )
   END_RUNG
   RUNG wire#w1
      Contact( "General_DB"."Bypass CIP Signal Homomixer" )
   END_RUNG wire#w4
   RUNG wire#w1
      I_Contact( "General_DB"."Bypass CIP Signal Homomixer" )
      Contact( "CIP_to_Mix".CIP_Complete.Homomixer."T-13.00_CIP_Complete" )
      Coil( "T-13.00_Homomixer"."CIP Complete" )
   END_RUNG
   // the same network as SCL:
   "T-13.00_Homomixer"."CIP Request OK" := "AlwaysTRUE" AND ((NOT "General_DB"."Bypass CIP Signal Homomixer" AND "CIP_to_Mix".CIP_RequestOK.Homomixer."T-13.00_CIP_RequestOK") OR "General_DB"."Bypass CIP Signal Homomixer");
   "T-13.00_Homomixer"."CIP In Progress" := "AlwaysTRUE" AND ((NOT "General_DB"."Bypass CIP Signal Homomixer" AND "CIP_to_Mix".CIP_InProgress.Homomixer."T-13.00_CIP_InProgress") OR "General_DB"."Bypass CIP Signal Homomixer");
   "T-13.00_Homomixer"."CIP Supply ON" := "AlwaysTRUE" AND ((NOT "General_DB"."Bypass CIP Signal Homomixer" AND "CIP_to_Mix".CIP_Supply_On.Homomixer."T-13.00_CIP_Supply_ON") OR "General_DB"."Bypass CIP Signal Homomixer");
   "T-13.00_Homomixer"."CIP Complete" := "AlwaysTRUE" AND NOT "General_DB"."Bypass CIP Signal Homomixer" AND "CIP_to_Mix".CIP_Complete.Homomixer."T-13.00_CIP_Complete";
END_REGION

REGION Network 26: T-14.00 DOSE ON OFF
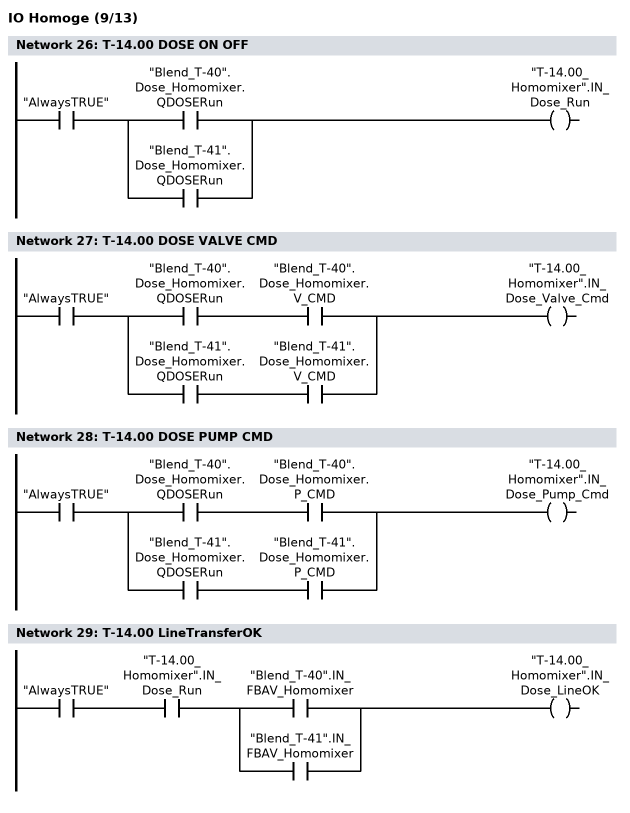
   RUNG wire#powerrail
      Contact( "AlwaysTRUE" )
      wire#w1
      Contact( "Blend_T-40".Dose_Homomixer.QDOSERun )
      wire#w2
      Coil( "T-14.00_Homomixer".IN_Dose_Run )
   END_RUNG
   RUNG wire#w1
      Contact( "Blend_T-41".Dose_Homomixer.QDOSERun )
   END_RUNG wire#w2
   // the same network as SCL:
   "T-14.00_Homomixer".IN_Dose_Run := "AlwaysTRUE" AND ("Blend_T-40".Dose_Homomixer.QDOSERun OR "Blend_T-41".Dose_Homomixer.QDOSERun);
END_REGION

REGION Network 27: T-14.00 DOSE VALVE CMD
   RUNG wire#powerrail
      Contact( "AlwaysTRUE" )
      wire#w1
      Contact( "Blend_T-40".Dose_Homomixer.QDOSERun )
      Contact( "Blend_T-40".Dose_Homomixer.V_CMD )
      wire#w2
      Coil( "T-14.00_Homomixer".IN_Dose_Valve_Cmd )
   END_RUNG
   RUNG wire#w1
      Contact( "Blend_T-41".Dose_Homomixer.QDOSERun )
      Contact( "Blend_T-41".Dose_Homomixer.V_CMD )
   END_RUNG wire#w2
   // the same network as SCL:
   "T-14.00_Homomixer".IN_Dose_Valve_Cmd := "AlwaysTRUE" AND (("Blend_T-40".Dose_Homomixer.QDOSERun AND "Blend_T-40".Dose_Homomixer.V_CMD) OR ("Blend_T-41".Dose_Homomixer.QDOSERun AND "Blend_T-41".Dose_Homomixer.V_CMD));
END_REGION

REGION Network 28: T-14.00 DOSE PUMP CMD
   RUNG wire#powerrail
      Contact( "AlwaysTRUE" )
      wire#w1
      Contact( "Blend_T-40".Dose_Homomixer.QDOSERun )
      Contact( "Blend_T-40".Dose_Homomixer.P_CMD )
      wire#w2
      Coil( "T-14.00_Homomixer".IN_Dose_Pump_Cmd )
   END_RUNG
   RUNG wire#w1
      Contact( "Blend_T-41".Dose_Homomixer.QDOSERun )
      Contact( "Blend_T-41".Dose_Homomixer.P_CMD )
   END_RUNG wire#w2
   // the same network as SCL:
   "T-14.00_Homomixer".IN_Dose_Pump_Cmd := "AlwaysTRUE" AND (("Blend_T-40".Dose_Homomixer.QDOSERun AND "Blend_T-40".Dose_Homomixer.P_CMD) OR ("Blend_T-41".Dose_Homomixer.QDOSERun AND "Blend_T-41".Dose_Homomixer.P_CMD));
END_REGION

REGION Network 29: T-14.00 LineTransferOK
   RUNG wire#powerrail
      Contact( "AlwaysTRUE" )
      Contact( "T-14.00_Homomixer".IN_Dose_Run )
      wire#w1
      Contact( "Blend_T-40".IN_FBAV_Homomixer )
      wire#w2
      Coil( "T-14.00_Homomixer".IN_Dose_LineOK )
   END_RUNG
   RUNG wire#w1
      Contact( "Blend_T-41".IN_FBAV_Homomixer )
   END_RUNG wire#w2
   // the same network as SCL:
   "T-14.00_Homomixer".IN_Dose_LineOK := "AlwaysTRUE" AND "T-14.00_Homomixer".IN_Dose_Run AND ("Blend_T-40".IN_FBAV_Homomixer OR "Blend_T-41".IN_FBAV_Homomixer);
END_REGION

REGION Network 30: T-14.00 Homomixer
